REGION Network 2: Block description — Sections 3.2 to 3.4
   // ▂▂▂▂▂▂▂▂▂▂▂▂▂▂▂▂▂▂▂▂▂▂▂▂▂▂▂▂▂▂▂▂▂▂▂▂▂▂▂▂▂▂▂▂
   // 3.2     Warnings and alarms
   // 
   // 
   // By default, the block generates 4 alarms and warnings (2 warnings and 2 alarms, 4 in total) 
   // as follows:
   // 
   // 
   //  ――――――――――――――――――――――――――――――――――――――――――
   //  ALARM / WARNING     FUNCTION
   //  ――――――――――――――――――――――――――――――――――――――――――
   //  Alarm high       Scaled signal is equal to or above a preset alarm high setpoint
   //  Warning high      Scaled signal is equal to or above a preset warning high setpoint
   //  Warning low     Scaled signal is equal to or below a preset warning low setpoint
   //  Alarm low      Scaled signal is equal to or below a preset alarm low setpoint
   //  ――――――――――――――――――――――――――――――――――――――――――
   //  Default alarm and warning signals
   // 
   // 
   // The active state of any alarm or warning is stored in the DYNAMIC_DATA structure in the following 
   // variables:
   // 
   // 
   //  UT22001_Dy_InstAnalogRead
   //  ――――――――――――――――――――――――――――――――――――――――――
   //  SIGNAL NAME          FUNCTION                     TYPE
   //  ――――――――――――――――――――――――――――――――――――――――――
   //  msg_Alm_H         MESSAGE — Alarm - high alarm is active        Bool
   //  msg_Alm_L          MESSAGE — Alarm - low alarm is active          Bool
   //  msg_Wrn_H          MESSAGE — Warning - high warning is active      Bool
   //  msg_Wrn_L          MESSAGE — Warning - low warning is active        Bool
   //  ――――――――――――――――――――――――――――――――――――――――――
   // 
   // 
   // The alarms and warnings that end with _H are activated when the scaled instrument reading is 
   // greater than or equal to a setpoint threshold (i.e. activate when the measured quantity is too 
   // high; generally, if there is both an alarm high and a warning high, the convention within the PAL 
   // is that the warning should activate before the alarm².
   // 
   // 
   // The alarms and warnings that end with _L are activated when the scaled instrument reading is 
   // less than or equal to a setpoint threshold (i.e. activate when the measured quantity is too low; 
   // generally, if there is both an alarm low and a warning low, the convention within the PAL is that 
   // the warning should activate before the alarm².
   // 
   // ――――――――――
   // ²         This is just a convention, there is nothing to stop the warning being set to occur after 
   //      the alarm (i.e. the warning detecting the most extreme condition). All alarms and 
   //      warnings are entirely independent of each other and no error checking is carried 
   //      out to ensure that any particular threshold is above or below another.
   // ――――――――――
   // 
   // All alarms and warnings are individually enabled (a disabled alarm or warning will never be 
   // activated), all alarms and warnings have individual setpoint values (the value at which the 
   // alarm or warning is triggered), all alarms and warnings have individual hysteresis valves 
   // (effectively a tolerance band, the difference between where an alarm activates and where it 
   // deactivates, used to prevent nuisance or “chattering” alarms). Finally, each alarm and warning 
   // has a configurable on and off delay (the alarm or warning will only activate if the reading is 
   // outside the threshold for the on-delay time and similarly will only deactivate when the reading 
   // is inside the threshold and hysteresis for the off-delay time).
   // 
   // The following table summarises all the available signals for each alarm and warning:
   // 
   // 
   //  ――――――――――――――――――――――――――――――――――――――――――
   //  SIGNAL          FUNCTION             TYPE   DETAILS
   //  ――――――――――――――――――――――――――――――――――――――――――
   //  CONFIG_XXX_Y_EN    Alarm/warning enabled      Bool    1 = enabled, 0 = disabled
   //  SP_XXX_Y_VAL      Alarm/warning setpoint value    Real Engineering units
   //  SP_XXX_Y_HYST_VAL    Alarm/warning hysteresis value Real Engineering units
   //  TIME_XXX_Y_ON_DEL   Alarm/warning on delay time   Real In seconds
   //  TIME_XXX_Y_OFF_DEL     Alarm/warning off delay time   Real In seconds
   //  mode_Xxx_Y_MaskOn     Alarm/warning is masked      Bool    1 = masked, 0 = normal
   //  msg_Xxx_Y         Alarm/warning is active      Bool    1 = active, 0 = inactive
   //  ――――――――――――――――――――――――――――――――――――――――――
   //  Default alarm and warning signals — where XXX is either ALM or WRN and Y is either H or L
   // 
   // 
   // 
   // ▁▁▁▁▁▁▁▁▁▁▁▁▁▁▁▁▁▁▁▁▁▁▁▁▁▁▁▁▁▁▁▁▁▁▁▁▁▁▁▁▁▁▁▁
   // 3.2.1     High alarms and warnings (an example)
   // 
   // 
   // This example explains how a high alarm signal is generated, a high warning works in exactly the 
   // same way with WRN being substituted for ALM.
   // 
   // The full set of signals associated with the high alarm are:
   // 
   // 
   //  ――――――――――――――――――――――――――――――――――――――――――
   //  SIGNAL           FUNCTION            TYPE   DETAILS
   //  ――――――――――――――――――――――――――――――――――――――――――
   //  CONFIG_ALM_H_EN    Alarm high enabled      Bool    1 = enabled, 0 = disabled
   //  SP_ALM_H_VAL      Alarm high setpoint value    Real Engineering units
   //  SP_ALM_H_HYST_VAL    Alarm high hysteresis value Real Engineering units
   //  TIME_ALM_H_ON_DEL   Alarm high on delay time   Real In seconds
   //  TIME_ALM_H_OFF_DEL     Alarm high off delay time   Real In seconds
   //  mode_Alm_H_MaskOn    Alarm is masked         Bool    1 = masked, 0 = normal
   //  msg_Alm_H        Alarm high is active      Bool    1 = active, 0 = inactive
   //  ――――――――――――――――――――――――――――――――――――――――――
   // 
   // 
   // The figure below indicates how each of these signal functions (note TIME_ALM_H_ON_DEL and
   // TIME_ALM_H_OFF_DEL have been abbreviated to ON_DEL and OFF_DEL respectively):
   // 
   // 
   //                 │
   //                 │          ╱╲╱╲
   //                 │    ①      ②╱    ╲
   //       SP_ALM_H_VAL↘│____╱╲________╱____________╲③_______④__________ 
   //    SP_ALM_H_HYST_VAL ↕│__╱____╲____╱╎_____╎_______╲____╱╲___________
   //                 │╱    ╲╱ ╎    ╎      ╲╱     ╲
   //                 │        ╎    ╎          ╎╲
   //                 │        ╎    ╎          ╎ ╲___
   //                 │        ╎    ╎          ╎    ╎╲╱
   //                 │    ON_DEL→╎    ╎←    OFF_DEL→╎    ╎←
   //                 ┼─────────────────────────────
   // 
   //                            ╎                        ╎
   // 
   //         msg_Alm_H │             ┏━━━━━━━━━━━━┓
   //                 │             ┃               ┃
   // CONFIG_ALM_H_EN = 1     │             ┃   ALARM IS ACTIVE    ┃
   // & mode_Alm_H_MaskOn = 0 │             ┃               ┃
   //                 │             ┃               ┃
   //                 ┼━━━━━━━━━━━━╶╶╶╶╶╶╶╶╶╶╶╶╶━━━━
   // 
   //                            ╎                        ╎
   // 
   //         msg_Alm_H │          
   // ⑤               │             ╎               ╎             
   // CONFIG_ALM_H_EN = 0     │             
   //     OR          │             ╎               ╎
   // CONFIG_ALM_H_EN = 1     │          
   // & mode_Alm_H_MaskOn = 1 ┼━━━━━━━━━━━━━━━━━━━━━━━━━━━━━
   // 
   // 
   // 
   // ▁▁▁▁▁▁▁▁▁▁▁▁▁▁▁▁▁▁▁▁▁▁▁▁▁▁▁▁▁▁▁▁▁▁▁▁▁▁▁▁▁▁▁▁
   // Scenario ①, alarm setpoint reached, but for less than on-delay duration
   // 
   // 
   // The graph represents the scaled analog instrument reading, actual_Value (in engineering 
   // units). The top horizontal line is the setpoint for the high alarm (SP_ALM_H_VAL).
   // 
   // If the alarm is enabled (CONFIG_ALM_H_EN = 1) then the following actions occur:
   // 
   // At point ① on the graph, the signal actual_Value reaches (and exceeds) the threshold value 
   // SP_ALM_H_VAL; i.e.:
   // 
   //           actual_Value ≥ SP_ALM_H_VAL
   // 
   // At this point, the alarm setpoint is exceeded and the on-delay timer starts; in the case of point ①, 
   // the signal actual_Value falls back below the setpoint value before the on-delay timer reaches 
   // the time set in TIME_ALM_H_ON_DEL, consequently the alarm does not activate.
   // 
   // 
   // 
   // ▁▁▁▁▁▁▁▁▁▁▁▁▁▁▁▁▁▁▁▁▁▁▁▁▁▁▁▁▁▁▁▁▁▁▁▁▁▁▁▁▁▁▁▁
   // Scenario ②, alarm setpoint reached for more than the on-delay duration
   // 
   // 
   // At point ② on the graph, the signal actual_Value again reaches (and exceeds) the setpoint value 
   // SP_ALM_H_VAL.
   // 
   // Again, at this point, the alarm threshold is exceeded and the on-delay timer starts; in the case of 
   // point ②, the signal actual_Value remains at or above the setpoint value for the full duration of 
   // the TIME_ALM_H_ON_DEL and consequently the alarm activates (msg_Alm_H goes to a high 
   // state), this is indicated in the middle msg_Alm_H graph.
   // 
   // 
   // 
   // ▁▁▁▁▁▁▁▁▁▁▁▁▁▁▁▁▁▁▁▁▁▁▁▁▁▁▁▁▁▁▁▁▁▁▁▁▁▁▁▁▁▁▁▁
   // Scenario ③, alarm reset level reached, but for less than the off-delay duration
   // 
   // 
   // At point ③, the signal actual_Value falls to the point at which the alarm is no longer active i.e.:
   // 
   //           actual_Value < (SP_ALM_H_VAL − SP_ALM_H_HYST_VAL)
   // 
   // Note:    in this case the inequality is less than (not less than or equal to), this is to prevent 
   //      conflict detecting the threshold and detecting the reset value if SP_ALM_H_HYST_VAL 
   //      is set to zero.
   // 
   // At this point, the signal is below the alarm reset level:
   // 
   //           SP_ALM_H_VAL − SP_ALM_H_HYST_VAL
   // 
   // and the off-delay timer starts; in the case of point ③, the signal actual_Value returns above the 
   // reset threshold before the off-delay timer reaches the time set in TIME_ALM_H_OFF_DEL, 
   // consequently, the alarm does not deactivate.
   // 
   // 
   // 
   // ▁▁▁▁▁▁▁▁▁▁▁▁▁▁▁▁▁▁▁▁▁▁▁▁▁▁▁▁▁▁▁▁▁▁▁▁▁▁▁▁▁▁▁▁
   // Scenario ④, alarm reset level reached for more than the off-delay duration
   // 
   // 
   // At point ④ on the graph, the signal actual_Value again falls below the alarm reset level 
   // (SP_ALM_H_VAL − SP_ALM_H_HYST_VAL).
   // 
   // Again, at this point, the off-delay timer starts; in the case of point ④, the signal actual_Value 
   // remains below the reset threshold for the full duration of the TIME_ALM_H_OFF_DEL and 
   // consequently, the alarm deactivates (msg_Alm_H goes to a low state), this is indicated in the 
   // middle msg_Alm_H graph.
   // 
   // 
   // 
   // ▁▁▁▁▁▁▁▁▁▁▁▁▁▁▁▁▁▁▁▁▁▁▁▁▁▁▁▁▁▁▁▁▁▁▁▁▁▁▁▁▁▁▁▁
   // Scenario ⑤, alarm is disabled
   // 
   // 
   // If the alarm is disabled (CONFIG_ALM_H_EN = 0) then the alarm will never activate 
   // (msg_Alm_H is always in a low state), this is indicated in the lower msg_Alm_H graph.
   // 
   // Note:    The timer for disabled alarms and warnings is permanently set to zero.
   // 
   // 
   // ▁▁▁▁▁▁▁▁▁▁▁▁▁▁▁▁▁▁▁▁▁▁▁▁▁▁▁▁▁▁▁▁▁▁▁▁▁▁▁▁▁▁▁▁
   // 3.2.2     Low alarms and warnings
   // 
   // 
   // Low alarms and warnings are very similar to the high alarms of § 3.2.1, they do however work
   // in the opposite sense (the inequalities are reversed), low alarms and warnings are activated
   // when the actual_Value falls below, or is equal to, the SP_ALM_L_VAL, and deactivates when it
   // rises above SP_ALM_L_VAL + SP_ALM_L_HYST_VAL.
   // 
   // On and off delays work in exactly the same way as those for the high alarm.
   // 
   // A worked example of the low alarm is given in the online documentation for this block:
   // 
   // select this block in the project tree and press:
   //      SHIFT + F1 or follow the link: https://psop.uk/pal-smds-fc02001-p
   // 
   // 
   // 
   // 
   // ▁▁▁▁▁▁▁▁▁▁▁▁▁▁▁▁▁▁▁▁▁▁▁▁▁▁▁▁▁▁▁▁▁▁▁▁▁▁▁▁▁▁▁▁
   // 3.2.3     Masking alarms and warnings
   // 
   // 
   // There are conditions where it can become necessary to mask (supress) alarms and warnings, a 
   // typical example could be a flow meter that monitors the flow into a filter; under normal 
   // conditions the flow meter would generate a low alarm if the flow into the filter were below a 
   // certain setpoint (indicating that the filter is becoming blocked).
   // 
   // It would be normal practice to supress this alarm when the filter was being cleaned, under 
   // these circumstances there would be no flow into the filter, but this would be a normal operating 
   // condition for the filter; the flow meter should only be monitoring for a low alarm during normal 
   // operation, not when the filter is being cleaned.
   // 
   // This suppression of an alarm or warning is referred to as “masking”, and there is a mask bit for 
   // each alarm and warning:
   // 
   // 
   //  ――――――――――――――――――――――――――――――――――――――――――
   //  SIGNAL           FUNCTION           TYPE   DETAILS
   //  ――――――――――――――――――――――――――――――――――――――――――
   //  mode_Alm_H_MaskOn    Masks the high alarm     Bool    1 = alarm masked, 0 = normal
   //  mode_Alm_L_MaskOn    Masks the low alarm    Bool    1 = alarm masked, 0 = normal
   //  mode_Wrn_H_MaskOn    Masks the high warning    Bool    1 = warning masked, 0 = normal
   //  mode_Wrn_L_MaskOn     Masks the low warning      Bool    1 = warning masked, 0 = normal
   //  ――――――――――――――――――――――――――――――――――――――――――
   //  Alarm and warning mask signals
   // 
   //  
   // Any alarm or warning that is masked (mode_Xxx_Y_MaskOn = 1), will deactivate instantly 
   // (there is no off-delay) and will not reactivate activate (the msg_Xxx_Y will be set to zero), the 
   // effect is the same as if the CONFIG_XXX_Y_EN bit were turned off.
   // 
   // The difference between the mask and the ENABLE signals is that the enable signal is a 
   // configuration of the instrument (it determines which alarms and warnings are configured for the 
   // particular instrument) and does not change at run-time (it is stored in static data block).
   // 
   // The mask signal on the other hand can be changed at run-time (either by some aspect of the 
   // Controller program or by the operator). The mask signal is stored in a dynamic data block and 
   // can be freely modified.
   // 
   // Note:    If an alarm or warning is not enabled (CONFIG_XXX_Y_EN = 0), then the mask bit 
   //      (mode_Xxx_Y_MaskOn) will not do anything (setting it will not enable the alarm), in 
   //      fact if the alarm or warning is not enabled, the mask bit will be permanently set to 
   //      zero.
   // 
   // Masking alarms and warnings is the correct way to disable an alarm as part of the process 
   // operation of the plant.
   // 
   // When an alarm or warning goes from a masked condition to an unmasked condition (returns to 
   // normal operation), the on-delay timer will be reset and any alarm or warning condition will 
   // have to go back through the on-delay process before the alarm or warning can reactivate, this is 
   // true even if the alarm were active before being masked.
   // 
   // 
   // 
   // 
   // ▁▁▁▁▁▁▁▁▁▁▁▁▁▁▁▁▁▁▁▁▁▁▁▁▁▁▁▁▁▁▁▁▁▁▁▁▁▁▁▁▁▁▁▁
   // 3.2.4     A note on dynamically enabling alarms
   // 
   // 
   // In normal operations, alarms are either enabled or disabled as part of the instrument 
   // configuration and this configuration will not change during run-time; the enable signal 
   // (CONFIG_XXX_Y_EN) is after all in a static data block. 
   // 
   // However, it is possible that the static data block is being used as a recipe block and as such it 
   // could be overloaded at some point during run-time.
   // 
   // Should the block detect a change in any of the CONFIG_XXX_Y_EN; specifically, a rising 
   // edge, the block provides error checking to ensure that the associated alarm/warning timer 
   // (actual_Xxx_Y_Timer) is preset to correct TIME_XXX_Y_ON_DEL, this prevents the alarm/warning 
   // from activating instantly, if the actual_Value is outside the alarm/warning setpoint. A condition 
   // that could arise because the timer is set to zero while ever the alarm/warning is disabled.
   // 
   // Note:    This is a minor technical point, but it is a necessary error trapping mechanism — the 
   //      situation could arise even if it is unlikely.
   // 
   // 
   // 
   // ▂▂▂▂▂▂▂▂▂▂▂▂▂▂▂▂▂▂▂▂▂▂▂▂▂▂▂▂▂▂▂▂▂▂▂▂▂▂▂▂▂▂▂▂
   // 3.3     Fault signals
   // 
   // 
   // There are four fault signals that can be produced by the block:
   // 
   // 
   //  ――――――――――――――――――――――――――――――――――――――――――
   //  SIGNAL           FUNCTION            TYPE   DETAILS
   //  ――――――――――――――――――――――――――――――――――――――――――
   //  msg_Flt_UnderRange   The instrument is more than   Bool    1 = under-range, 0 = healthy
   //                 a percentage below the its 
   //                 minimum value
   // 
   //  msg_Flt_OverRange     The instrument is more than   Bool    1 = over-range, 0 = healthy
   //                 a percentage above its 
   //                 maximum value
   // 
   //  msg_Flt_OutOfRange   Common fault, either       Bool    1 = out-of-range, 0 = healthy
   //                 under or over range
   // 
   //  msg_Flt_External     The instrument itself is    Bool    1 = fault, 0 = healthy
   //                 indicating a fault 
   //                 (hardwired signal)
   //  ――――――――――――――――――――――――――――――――――――――――――
   //  Block fault signals 
   // 
   // 
   // 
   // ▁▁▁▁▁▁▁▁▁▁▁▁▁▁▁▁▁▁▁▁▁▁▁▁▁▁▁▁▁▁▁▁▁▁▁▁▁▁▁▁▁▁▁▁
   // 3.3.1     Over, under and out of range fault signals
   // 
   // If the scaled signal actual_Value , is outside the RANGE_SCALE_MIN to RANGE_SCALE_MAX range 
   // (dotted area of the graph, § 3.1), the scaled instrument reading (actual_Value) will still be 
   // calculated correctly; however, an appropriate, over-range or under-range (msg_Flt_OverRange or 
   // msg_Flt_UnderRange) signal will be generated to indicate that the instrument signal is outside 
   // of its calibrated range and is potentially no longer accurate.
   // 
   // Some tolerance is permitted before either the msg_Flt_OverRange or msg_Flt_UnderRange 
   // signals is activated (this is to prevent nuisance alarms — most instruments are tolerant of slight 
   // over and under shoot readings). 
   // 
   // The tolerance applied to the out-of-range signals is a percentage of the scaled range of the 
   // instrument (the scaled range being RANGE_SCALE_MAX − RANGE_SCALE_MIN). 
   // 
   // The tolerance to be applied is given in the parameter RANGE_OOR_PERCENT, this is a real 
   // (floating point) number in the range 0.0-10.0%.
   // 
   // If the tolerance for the instrument is not known, a generic value of 2.5% should be used.
   // 
   // The out-of-range tolerance absolute value (in terms of the actual_Value rather than as a 
   // percentage) is calculated as:
   // 
   // 
   // ┌───────────────────────────────────────┐
   // │                            (RANGE_SCALE_MAX ─ RANGE_SCALE_MIN) ╳ RANGE_OOR_PERCENT  │
   // │ calAbsOOR =  ――――――――――――――――――――――――――――――    │
   // │                        100                 │
   // └───────────────────────────────────────┘
   // 
   // 
   // Thus, if RANGE_SCALE_MIN is −100 l/s, RANGE_SCALE_MAX is +100 l/s (giving a span of 200 l/s) and 
   // a RANGE_OOR_PERCENT of 2.5% is selected, the absolute out of range value (calAbsOOR in the 
   // above equation) has a calculated value of 5.00 l/s (2.5% of 200).
   // 
   // In this example, the msg_Flt_OverRange signal would activate when actual_Value exceeded a 
   // value of RANGE_SCALE_MAX + 5.00 (or 105.00  l/s). This value (the absolute over range limit 
   // value) is stored in a calculated variable cal_OR_Abs. 
   // 
   // Similarly, the msg_Flt_UnderRange signal would activate when actual_Value fell below a value 
   // of RANGE_SCALE_MIN – 5.00 (or −105.00  l/s). This value (the absolute under range limit value) 
   // is stored in a calculated variable cal_UR_Abs.
   // 
   // Both the cal_OR_Abs and cal_UR_Abs values are stored in  the dynamic data area and can be 
   // accessed by SCADA and HMI systems, or other aspects of the Con-troller software.
   // 
   // 
   // 
   // ▁▁▁▁▁▁▁▁▁▁▁▁▁▁▁▁▁▁▁▁▁▁▁▁▁▁▁▁▁▁▁▁▁▁▁▁▁▁▁▁▁▁▁▁
   // Common out of range signal
   // 
   // 
   // There is a third out of range signal: msg_Flt_OutOfRange, this signal is a common signal that 
   // just indicates the instrument is out of its calibrated range (it does not specify whether it is over 
   // or under range). It is activated if either the msg_Flt_OverRange or msg_Flt_UnderRange signal is 
   // active.
   // 
   // 
   // 
   // ▁▁▁▁▁▁▁▁▁▁▁▁▁▁▁▁▁▁▁▁▁▁▁▁▁▁▁▁▁▁▁▁▁▁▁▁▁▁▁▁▁▁▁▁
   // Configuration error
   // 
   // If a range configuration error is present (see § 3.1.2), all three out of range signals will activate 
   // msg_Flt_OverRange, msg_Flt_UnderRange and msg_Flt_OutOfRange.
   // 
   // 
   // 
   // ▁▁▁▁▁▁▁▁▁▁▁▁▁▁▁▁▁▁▁▁▁▁▁▁▁▁▁▁▁▁▁▁▁▁▁▁▁▁▁▁▁▁▁▁
   // 3.3.2     External fault signal
   // 
   // 
   // The external fault is an optional hardwired signal from the instrument, it indicates that the 
   // instrument itself is registering that there is some problem. Such external fault signals are more 
   // commonly associated with complex instruments (mass flow metres, ultrasonic level 
   // transducers, analytical instruments &c.) rather than the more simplistic instruments (pressure 
   // sensors, temperature transmitters &c.).
   // 
   // Typical examples of external faults would be:
   // 
   //    •   No medium present in a mass flow meter (if the instrument were measuring liquid 
   //      flow and the pipe had become empty)
   // 
   //    •   Foam indication from an ultrasonic level transducer (preventing an accurate level 
   //      reading)
   // 
   // Such fault signals are generally indicated via a hardwired digital input to the Controller.
   // 
   // The external fault signal (if used) is passed to the block as the parameter: EXT_FAULT
   // 
   // 
   //  ――――――――――――――――――――――――――――――――――――――――――
   //  PARAMETER          FUNCTION            TYPE   DETAILS
   //  ――――――――――――――――――――――――――――――――――――――――――
   //  EXT_FAULT        Hardwired signal indicating    Bool    1 = fault, 0 = healthy
   //                 the instrument is in a fault 
   //                 condition
   //  ――――――――――――――――――――――――――――――――――――――――――
   //  Block external fault parameter 
   // 
   // 
   // If the EXT_FAULT signal is not required, the input should be set to _false.
   // 
   // If the instrument generates a fault signal in the opposite sense, i.e. 0 = fault and 1 = healthy (this 
   // is a common fail-safe condition, that generates a fault signal if the instrument is disconnected 
   // or a wire break occurs), then a normally closed contact should be applied to the EXT_FAULT 
   // parameter to invert the signal into the block (see below):
   // 
   // 
   //                            ┌─────────────
   //         ───────────────────┤ FC02001 
   //                            │               │                       
   //                                "FC001" ─┤ AI_RAW_SIGNAL          │
   //                            │               │
   //       "DB00801_St_ConstAiRawData".AI_RAW_2003 ─┤ AI_RAW_DATA           │
   //                            │               │
   //    "DB00851_St_ConstAiScaleData".AI_SCALE_FC001    ─┤ AI_SCALE_DATA          │
   //                            │               │
   //              "FC001_FAULT"           │               │
   //           ────┤╱├──────────┤ EXT_FAULT                │
   //                            │               │
   //                            │               │
   //         "DB02001_St_StdInstAnalogRead".FC001 ─┤ STATIC_DATA             │
   //                            │
   //        "DB22001_Dy_StdInstAnalogRead".FC001 ─┤ DYNAMIC_DATA
   //                            │
   //                            │
   // 
   // 
   // If the EXT_FAULT parameter is activated (set to 1), the corresponding fault signal within the 
   // dynamic data (msg_Flt_External) will be activated, there are no delays or other filtering 
   // associated with this signal.
   // 
   // Note:    The external fault does not in any way impact the reading and scaling of the 
   //      instrument or the production of any alarms or warnings.
   // 
   // 
   // 
   // ▂▂▂▂▂▂▂▂▂▂▂▂▂▂▂▂▂▂▂▂▂▂▂▂▂▂▂▂▂▂▂▂▂▂▂▂▂▂▂▂▂▂▂▂
   // 3.4     Operating mode
   // 
   // 
   // This block  supports various operating modes:
   // 
   //    •   Simulation mode
   //    •   Remote/local mode
   //    •   Faceplate disabled mode
   // 
   // Examining these in turn:
   // 
   // 
   // ▁▁▁▁▁▁▁▁▁▁▁▁▁▁▁▁▁▁▁▁▁▁▁▁▁▁▁▁▁▁▁▁▁▁▁▁▁▁▁▁▁▁▁▁
   // 3.4.1     Simulation mode
   // 
   // 
   // The instrument can be switched to a simulation mode, in which the actual reading from the 
   // instrument is replaced by a simulated value provided by the operator. 
   // 
   // Simulation mode is generally used during testing, but can also be applied in a process 
   // environment if a fault condition is detected within the instrument; this scenario allows the plant 
   // to continue operating (albeit under some degree of manual control) until the instrument is 
   // repaired or replaced.
   // 
   // The following data points are associated with the simulation mode:
   // 
   // 
   //  ――――――――――――――――――――――――――――――――――――――――――
   //  SIGNAL           FUNCTION            TYPE   DETAILS
   //  ――――――――――――――――――――――――――――――――――――――――――
   //  CONFIG_SIM_DIS         Prevents simulation mode   Bool    1 = no sim, 0 = sim permitted
   //                 being activated under all 
   //                 circumstances
   // 
   //  mode_SimOn        Activates simulation mode,    Bool    1 = sim on, 0 = sim off
   //                 if active, the scaled reading 
   //                 of the instrument:
   //                 actual_Value will be set 
   //                 to mode_SimValue
   // 
   //  mode_SimValue      Scaled instrument reading   Real    Simulated instrument value
   //                 actual_Value will be set to  
   //                 this if simulation mode is 
   //                 on (CONFIG_SIM_DIS = 0 
   //                 and mode_SimOn = 1)
   // 
   //  status_SimOn       Status indication, shows if    Bool    1 = sim active, 0 = Sim off
   //                 simulation mode is active
   //  ――――――――――――――――――――――――――――――――――――――――――
   // 
   // 
   // Simulation mode can only be activated by the operator via a faceplate available at the 
   // supervisory system (SCADA/HMI).
   // 
   // If simulation mode is disabled (configuration signal CONFIG_SIM_DIS is set to 1), then the 
   // simulation mode cannot be turned on under any circumstances, the option is greyed out on the 
   // supervisory system faceplate and the block will constantly reset the mode_SimOn signal.
   // 
   // If simulation mode is permitted (CONFIG_SIM_DIS = 0), then setting mode_SimOn to 1 will 
   // activate simulation mode and the scaled instrument value (actual_Value) will be set to the 
   // value stored in mode_SimValue:
   // 
   //           i.e. actual_Value = mode_SimValue
   // 
   // and all fault messages will be reset.
   // 
   // The operator can set and adjust the simulation value (mode_SimValue) from the instrument
   // faceplate on the supervisory system. The simulation value can be adjusted at any time by the 
   // operator (even if simulation mode has not been activated), but will not be applied until 
   // simulation mode is turned on (mode_SimOn = 1). 
   // 
   // If simulation mode is completely disabled (CONFIG_SIM_DIS is set to 1) then the operator will
   // not be able to adjust the simulated value (mode_SimValue will be greyed out on the faceplate).
   // 
   // 
   // 
   // ▁▁▁▁▁▁▁▁▁▁▁▁▁▁▁▁▁▁▁▁▁▁▁▁▁▁▁▁▁▁▁▁▁▁▁▁▁▁▁▁▁▁▁▁
   // 3.4.2     Remote/local mode
   // 
   // 
   // Remote and local operating modes refer to the supervisory system that has control of the 
   // instrument (i.e. which system can write to the device and change the operating mode of the 
   // device). 
   // 
   // This type of mode is usual present where a plant has a remote central control location (a control 
   // room) that normally controls the device (remote control), but also has a field panel with a local 
   // HMI that an operator in the field can select to take over control of the device (local control) for 
   // maintenance purposes.
   // 
   // The modes are as follows (and are mutually exclusive, only one will be active):
   // 
   //    Remote        Only the remote system in the control room can 
   //                 control the device
   // 
   //    Local            A local system has taken control of the device and the remote 
   //                 system can no longer issue commands to it
   // 
   //    Remote/local disabled   The system does not use remote/local modes and any 
   //    (ALL mode)       supervisory system can issue commands to the device 
   //  
   // Remote/local control is generally handled by the supervisory systems themselves; however, the 
   // supervisory systems need a storage area per device to record which mode that device is in, local 
   // control is often activated by a panel key-switch, that changes the state of several devices from 
   // remote to local (usually all the devices controlled by the local panel).
   // 
   // The block simply identifies the remote/local mode from the mode signals and configuration 
   // signals provided to the block.
   // 
   // For systems that do not use remote/local modes (any supervisory system can control the device, 
   // or control is determined by operator privileges), the remote/local modes can be disabled 
   // (CONFIG_RL_EN is set to zero) and the device is effectively in ALL mode (any system can 
   // control the device).
   // 
   // If remote/local operation is in use, the supervisory system that does not have control will still 
   // display all the information from the device, but will not be able to control the device (it could not 
   // for example, activate simulation mode) and all control function (faceplate functions) will be 
   // greyed out.
   // 
   // The following signals are associated with remote/local/all modes:
   // 
   // 
   //  ――――――――――――――――――――――――――――――――――――――――――
   //  SIGNAL           FUNCTION            TYPE   DETAILS
   //  ――――――――――――――――――――――――――――――――――――――――――
   //  CONFIG_RL_EN      Allows Remote and Local      Bool    1 = Remote/local selected
   //                 modes to be selected        0 = All mode is active
   // 
   //  mode_RemoteOn       Activates remote mode     Bool    1 = remote mode on, 
   //                 CONFIG_RL_EN must = 1       0 = remote mode off
   // 
   //  mode_LocalOn     Activates local mode          Bool    1 = local mode on, 
   //                 CONFIG_RL_EN must = 1       0 = remote mode off
   // 
   //  status_RemoteOn      Status remote mode on     Bool    1 = remote mode on, 
   //                               0 = remote mode off
   // 
   //  status_LocalOn       Status local mode on      Bool    1 = local mode on, 
   //                               0 = local mode off
   // 
   //  status_RLOff       Status Remote/local is off     Bool    1 = ALL mode on, 
   //              (ALL mode active)         0 = ALL mode off
   //  ――――――――――――――――――――――――――――――――――――――――――
   //  Block remote/local signals 
   // 
   // 
   // By default, remote/local is disabled — ALL mode is selected (CONFIG_RL_EN = 0).
   // 
   // 
   // 
   // 
   // ▁▁▁▁▁▁▁▁▁▁▁▁▁▁▁▁▁▁▁▁▁▁▁▁▁▁▁▁▁▁▁▁▁▁▁▁▁▁▁▁▁▁▁▁
   // 3.4.3     Faceplate disable mode
   // 
   // 
   // It is possible to disable the supervisory system faceplate from within the block, the configuration 
   // signal:
   // 
   // 
   //  ――――――――――――――――――――――――――――――――――――――――――
   //  SIGNAL           FUNCTION            TYPE   DETAILS
   //  ――――――――――――――――――――――――――――――――――――――――――
   //  CONFIG_FP_DIS        Disable the supervisory      Bool    1 = Faceplate disabled
   //                 system faceplate           0 = normal
   //  ――――――――――――――――――――――――――――――――――――――――――
   //  Block faceplate disable signal 
   // 
   // 
   // If the faceplate is disabled (CONFIG_FP_DIS = 1), the supervisory system will not allow the 
   // device faceplate to be opened (normally achieved by clicking the block icon or device symbol), 
   // this in turn prevents the operator from affecting the device in anyway, it would not, for example, 
   // be possible to put the device into simulation mode.
END_REGION

REGION Network 3: Block description — Sections 3.5 to 11
   // ▂▂▂▂▂▂▂▂▂▂▂▂▂▂▂▂▂▂▂▂▂▂▂▂▂▂▂▂▂▂▂▂▂▂▂▂▂▂▂▂▂▂▂▂
   // 3.5     Status reporting
   // 
   // The module constantly reports the status of the instrument (i.e. alarm/warning states, faults &c.) 
   // via various status signals. These signals can be used within the Controller software to determine 
   // specific device conditions (e.g. a high alarm is active), the signals may also be used by 
   // supervisory systems to display (in an ani-mated fashion) the state of the instrument.
   // 
   // The status signals for faults, alarms and warnings are either duplicates of the message signals 
   // (signals beginning with msg_) or logical combinations of them.
   // 
   // The following is a full list of the status signals:
   // 
   // 
   //  UT22001_Dy_InstAnalogRead
   //  ――――――――――――――――――――――――――――――――――――――――――
   //  SIGNAL           FUNCTION            TYPE   DETAILS
   //  ――――――――――――――――――――――――――――――――――――――――――
   //  status_Alm_H        Identical to: msg_Alm_H    Bool    1 = high alm active, 0 = no alm
   // 
   //  status_Alm_L         Identical to: msg_Alm_L       Bool    1 = low alm active, 0 = no alm
   // 
   //  status_Wrn_H        Identical to: msg_Wrn_H    Bool    1 = high wrn active, 0 = no wrn
   // 
   //  status_Wrn_L         Identical to: msg_Wrn_L     Bool    1 = low wrn active, 0 = no wrn
   // 
   //  status_Alm_H_Mask     High alarm is masked     Bool    1 = masked, 0 = normal
   // 
   //  status_Alm_L_Mask   Low alarm is masked      Bool    1 = masked, 0 = normal
   // 
   //  status_Wrn_H_Mask      High warning is masked    Bool    1 = masked, 0 = normal
   // 
   //  status_Wrn_L_Mask       Low warning is masked     Bool    1 = masked, 0 = normal
   // 
   //  status_Alm_H_Dis         High alarm is disabled       Bool    1 = disabled, 0 = normal
   // 
   //  status_Alm_L_Dis       Low alarm is disabled        Bool    1 = disabled, 0 = normal
   // 
   //  status_Wrn_H_Dis          High warning is disabled      Bool    1 = disabled, 0 = normal
   // 
   //  status_Wrn_L_Dis           Low warning is disabled       Bool    1 = disabled, 0 = normal
   // 
   //  status_Fault       Indicates any of the msg_Flt    Bool    1 = fault active, 0 = healthy
   //                 signals are active:
   //                  msg_Flt_UnderRange
   //                  msg_Flt_OverRange
   //                  msg_Flt_OutOfRange
   //                  msg_Flt_External 
   // 
   //  status_SimOn       Status simulation mode on     Bool    1 = sim on, 0 = sim off
   // 
   //  status_RemoteOn      Status remote mode on     Bool    1 = rem on, 0 = rem off
   // 
   //  status_LocalOn       Status local mode on      Bool    1 = loc on, 0 = loc off 
   // 
   //  status_RLOff       Status ALL mode is on           Bool    1 = ALL mode on, 
   //                               0 = ALL mode off
   //  ――――――――――――――――――――――――――――――――――――――――――
   //  Block status signals 
   // 
   // 
   // 
   // ▁▁▁▁▁▁▁▁▁▁▁▁▁▁▁▁▁▁▁▁▁▁▁▁▁▁▁▁▁▁▁▁▁▁▁▁▁▁▁▁▁▁▁▁
   // 3.5.1     String constants for tag name and units
   // 
   // 
   // The STATIC_DATA structure holds two string values:
   // 
   // 
   //  UT02001_St_InstAnalogRead
   //  ――――――――――――――――――――――――――――――――――――――――――
   //  SIGNAL NAME          FUNCTION                     TYPE
   //  ――――――――――――――――――――――――――――――――――――――――――
   //  INFO_TAG          INFORMATION — Instrument ID tag          String[20]
   // 
   //  INFO_UNITS          INFORMATION — Instrument engineering units       String[10]
   //                        (unit of measure)
   //  ――――――――――――――――――――――――――――――――――――――――――
   //  String constants for the instrument
   // 
   // 
   // These two strings allow the supervisory system to populate the instrument tag (e.g. FIC001) and 
   // the engineering units applicable to the instrument (L/s for example) directly from the data 
   // stored in the PLC; it means the block icon can be used directly within the supervisory system 
   // graphic without customisation; all the data will be populated directly at runtime.
   // 
   //                ━━━   ⬙⬙⬙⬙⬙⬙   ━━━
   // 
   // 
   // 
   // ▄▄▄▄▄▄▄▄▄▄▄▄▄▄▄▄▄▄▄▄▄▄▄▄▄▄▄▄▄▄▄▄▄▄▄▄▄▄▄▄▄▄▄▄
   // 4.     Supervisory system interface
   // 
   // 
   // See the online documentation for this block — select the block in the project tree and press:
   //      SHIFT + F1 or follow the link: https://psop.uk/pal-smds-fc02001-p 
   // 
   // An explanation of the block icons and faceplates available to the supervisory system for this 
   // module is given in section 4 of the SMDS document [Ref. 011].
   // 
   // A downloadable copy of the SMDS (and all other project documentation) is available here:
   // 
   //      https://practicalseries.com/2001-pal/21-project/01-00-docs.html
   // 
   // For this module, the document number is: PS2001-5-2312-fc02001
   // 
   //                ━━━   ⬙⬙⬙⬙⬙⬙   ━━━
   // 
   // 
   // 
   // ▄▄▄▄▄▄▄▄▄▄▄▄▄▄▄▄▄▄▄▄▄▄▄▄▄▄▄▄▄▄▄▄▄▄▄▄▄▄▄▄▄▄▄▄
   // 5.     PARAMETERS
   // 
   // 
   // The following parameters are associated with the block:
   // 
   //  
   //  ――――――――――――――――――――――――――――――――――――――――――
   //  PARAM         FUNCTION                      TYPE      IN-OUT 
   //  ――――――――――――――――――――――――――――――――――――――――――
   //  SYS_SIGNALS      Common system signals                UT21000    In
   //           logic and timing signals for parametric access
   // 
   //  AI_RAW_SIGNAL      The unscaled analog input (input word          Word     In
   //           address for the IO card to which the instrument 
   //           is connected)
   //  AI_RAW_DATA      Analog input signal configuration data (type,     UT00801    In
   //           range, descriptions card parameters and 
   //           coefficients)
   // 
   //  AI_SCALE_DATA     Analog input signal scaled value data (instrument   UT00851   In
   //           tag, range, descriptions and engineering units)
   // 
   // 
   //  EXT_FAULT     Optional external fault signal for the instrument     Bool      In
   //           (1 = fault, 0 = healthy). If not required, set 
   //           permanently to _False
   // 
   //  STATIC_DATA     Data structure that holds the configuration data    UT02001    In
   //           for the instrument (raw range, scaled range 
   //           alarm and warning values, filtering times, 
   //           hysteresis values &c.)
   // 
   //  DYNAMIC_DATA      Data structure that holds the live data for the      UT22001    InOut
   //           instrument (its reading in engineering units, 
   //           any alarms or warnings that may be active, 
   //           current timer values, selected operating 
   //           mode &c.)
   //  ――――――――――――――――――――――――――――――――――――――――――
   // 
   // 
   //                ━━━   ⬙⬙⬙⬙⬙⬙   ━━━
   // 
   // 
   // 
   // ▄▄▄▄▄▄▄▄▄▄▄▄▄▄▄▄▄▄▄▄▄▄▄▄▄▄▄▄▄▄▄▄▄▄▄▄▄▄▄▄▄▄▄▄
   // 6.     DATA STRUCTURES AND USAGE
   // 
   // 
   // The block has the following associated data structure:
   // 
   // 
   //  ――――――――――――――――――――――――――――――――――――――――――
   //  DATA STRUCTURE             DESCRIPTION
   //  ――――――――――――――――――――――――――――――――――――――――――
   //  UT01000_St_SysRevision          Revision information for this block    See FC01001
   //  UT01001_St_SysLicence           Licence information for this block  See FC01001
   //  UT21000_Dy_SysSignals           System signals for logic and timing  See FC01001
   // 
   //  UT00801_St_ConstAiRawData        Analog input signal configuration data 
   //                     (type, range, descriptions card parameters and 
   //                     coefficients)
   // 
   //  UT00851_St_ConstAiScaleData     Analog input signal scaled value data 
   //                     (instrument tag, range, descriptions and 
   //                     engineering units)
   // 
   //  UT02001_St_InstAnalogRead      Static data structure for an analog instrument.
   //                     Holds configuration information, instrument ranges 
   //                     and scaling, alarm/warning thresholds &c.
   // 
   //  UT22001_Dy_InstAnalogRead        Dynamic data structure for an analog instrument.
   //                     Current scaled instrument reading, alarm status, 
   //                     operating modes, timer values &c.
   //  ――――――――――――――――――――――――――――――――――――――――――
   // 
   // 
   // 
   // ▂▂▂▂▂▂▂▂▂▂▂▂▂▂▂▂▂▂▂▂▂▂▂▂▂▂▂▂▂▂▂▂▂▂▂▂▂▂▂▂▂▂▂▂
   // 6.1     UT00801_St_ConstAiRawData
   // 
   // 
   // The static data structure for an analog instrument.
   // 
   // 
   //  UT00801_St_ConstAiRawData (full contents)
   //  ―――――――――――――――――――――――――――――――――――――――――― 
   //  SIGNAL NAME          FUNCTION                     TYPE
   //  ――――――――――――――――――――――――――――――――――――――――――
   //  AI_CODE            A 16-bit hex value that uniquely identifies dataset   UInt
   //               (it is the variable name of the dataset in DB00801)
   //  RAW_MIN         Minimum value of the raw analog signal        Int
   //               (at the card)
   // 
   //  RAW_MAX           Maximum value of the raw analog signal        Int
   //  RAW_DESC         Textual plain English description of the channel     String[60]
   //               type and range
   //  PARAM_TYPE         An 8-bit hex code that represents the input type    Byte
   //               See [Ref. 101]
   // 
   //  PARAM_RANGE        An 8-bit hex code that represents the input range    Byte
   //               See [Ref. 101]
   // 
   //  PARAM_COEF        An 8-bit hex code that represents a thermal        Byte
   //               coefficient (thermal resistance channels only, 
   //               otherwise set to 0). See [Ref. 101]
   // 
   //  VALUE_COEF        The actual value of the temperature coefficient in    Real
   //               use (thermal resistance channels only)
   //  ―――――――――――――――――――――――――――――――――――――――――― 
   // 
   // 
   // 
   // ▂▂▂▂▂▂▂▂▂▂▂▂▂▂▂▂▂▂▂▂▂▂▂▂▂▂▂▂▂▂▂▂▂▂▂▂▂▂▂▂▂▂▂▂
   // 6.2     UT00851_St_ConstAiScaleData
   // 
   // 
   // The static data structure for an analog instrument.
   // 
   // 
   //  UT00801_St_ConstAiRawData (full contents)
   //  ―――――――――――――――――――――――――――――――――――――――――― 
   //  SIGNAL NAME          FUNCTION                     TYPE
   //  ――――――――――――――――――――――――――――――――――――――――――
   //  AI_TAG          Tag name of the instrument             UInt
   //  SCALE_MIN        Minimum value of the scaled input signal range    Real
   //               being used by the module
   //  SCALE_MAX          Maximum value of the scaled input signal range      Real
   //               being used by the module
   //  SCALE_UNITS          Engineering units for the instrument         String[20]
   //  SCALE_DESC           Textual plain English description of the instrument  String[60]
   // 
   //  ―――――――――――――――――――――――――――――――――――――――――― 
   // 
   // 
   // 
   // ▂▂▂▂▂▂▂▂▂▂▂▂▂▂▂▂▂▂▂▂▂▂▂▂▂▂▂▂▂▂▂▂▂▂▂▂▂▂▂▂▂▂▂▂
   // 6.3     UT02001_St_InstAnalogRead
   // 
   // 
   // The static data structure for an analog instrument.
   // 
   // 
   //  UT02001_St_InstAnalogRead (full contents)
   //  ―――――――――――――――――――――――――――――――――――――――――― 
   //  SIGNAL NAME          FUNCTION                     TYPE
   //  ―――――――――――――――――――――――――――――――――――――――――― 
   //  CONFIG_ALM_H_EN     CONFIG — High alarm is enabled          Bool
   //                      (1 = enabled, 0 = no alarm) 
   //  CONFIG_ALM_L_EN      CONFIG — Low alarm is enabled           Bool
   //                      (1 = enabled, 0 = no alarm)
   //  CONFIG_WRN_H_EN        CONFIG — High warning is enabled         Bool
   //                      (1 = enabled, 0 = no warning)
   //  CONFIG_WRN_L_EN        CONFIG — Low warning is enabled          Bool
   //                      (1 = enabled, 0 = no warning)
   //  CONFIG_FP_DIS         CONFIG — Faceplate is disabled           Bool
   //                      (1 = no Faceplate, 0 = normal)
   //  CONFIG_SIM_DIS       CONFIG — Simulation is disabled            Bool
   //                      (1 = no Simulation, 0 = normal)
   //  CONFIG_RL_EN       CONFIG — Remote/local mode enabled       Bool
   //                      (1 = enabled, 0 = all mode)
   // 
   //  RANGE_RAW_MIN       RANGE — Minimum value of the raw analog      Int
   //                     signal (at the card). Only used if 
   //                     AI_RAW_DATA is set to User Defined input 
   //                     (AI_CODE = 0000)
   //  RANGE_RAW_MAX      RANGE — Maximum value of the raw analog        Int
   //                     signal (at the card). Only used if 
   //                     AI_RAW_DATA is set to User Defined input 
   //                     (AI_CODE = 0000)
   //  RANGE_OOR_PERCENT      RANGE — Out of range percentage, beyond which    Real
   //                     the instrument is out of range
   // 
   //  SP_ALM_H_VAL       SETPOINT — High alarm threshold value         Real
   //                      [engineering units]
   //  SP_ALM_L_VAL       SETPOINT — Low alarm threshold value       Real
   //                      [engineering units]
   //  SP_WRN_H_VAL         SETPOINT — High warning threshold value        Real
   //                      [engineering units]
   //  SP_WRN_L_VAL       SETPOINT — Low warning threshold value      Real
   //                      [engineering units]
   //  SP_ALM_H_HYST_VAL     SETPOINT — High alarm hysteresis value        Real
   //                      [engineering units]
   //  SP_ALM_L_HYST_VAL     SETPOINT — Low alarm hysteresis value         Real
   //                      [engineering units]
   //  SP_WRN_H_HYST_VAL    SETPOINT — High warning hysteresis value       Real
   //                      [engineering units]
   //  SP_WRN_L_HYST_VAL     SETPOINT — Low warning hysteresis value        Real
   //                      [engineering units]
   // 
   //  TIME_ALM_H_ON_DEL    TIMER — High alarm on delay time          Real
   //                      (activation delay), [seconds]
   //  TIME_ALM_L_ON_DEL     TIMER — Low alarm on delay time           Real
   //                      (activation delay), [seconds]
   //  TIME_WRN_H_ON_DEL       TIMER — High warning on delay time         Real
   //                      (activation delay), [seconds]
   //  TIME_WRN_L_ON_DEL        TIMER — Low warning on delay time          Real
   //                      (activation delay), [seconds]
   //  TIME_ALM_H_OFF_DEL      TIMER — High alarm off delay time           Real
   //                      (deactivation delay), [seconds]
   //  TIME_ALM_L_OFF_DEL       TIMER — Low alarm off delay time            Real
   //                      (deactivation delay), [seconds]
   //  TIME_WRN_H_OFF_DEL      TIMER — High warning off delay time          Real
   //                      (deactivation delay), [seconds]
   //  TIME_WRN_L_OFF_DEL      TIMER — Low warning off delay time           Real
   //                      (deactivation delay), [seconds]
   //  ――――――――――――――――――――――――――――――――――――――――――
   // 
   // 
   // 
   // ▂▂▂▂▂▂▂▂▂▂▂▂▂▂▂▂▂▂▂▂▂▂▂▂▂▂▂▂▂▂▂▂▂▂▂▂▂▂▂▂▂▂▂▂
   // 6.4      UT22001_Dy_InstAnalogRead
   // 
   // 
   // The static data structure for an analog instrument.
   // 
   // 
   //  UT22001_Dy_InstAnalogReadl (full contents)
   //  ――――――――――――――――――――――――――――――――――――――――――
   //  SIGNAL NAME          FUNCTION                     TYPE
   //  ――――――――――――――――――――――――――――――――――――――――――
   //  status_ConfigError       STATUS — Raw or scaled range configuration error   Bool
   //                      (1 = Config error, 0 = OK)
   //  status_Alm_H         STATUS — High alarm is active           Bool
   //                      (1 = alarm active, 0 = no alarm)
   //  status_Alm_L          STATUS — Low alarm is active            Bool
   //                      (1 = alarm active, 0 = no alarm)
   //  status_Wrn_H         STATUS — High warning is active          Bool
   //                      (1 = warning active, 0 = no warning)
   //  status_Wrn_L          STATUS — Low warning is active           Bool
   //                      (1 = warning active, 0 = no warning)
   //  status_Alm_H_Mask       STATUS — High alarm is masked             Bool
   //                      (1 = alarm masked, 0 = normal)
   //  status_Alm_L_Mask        STATUS — Low alarm is masked              Bool
   //                      (1 = alarm masked, 0 = normal)
   //  status_Wrn_H_Mask       STATUS — High warning is masked            Bool
   //                      (1 = warning masked, 0 = normal)
   //  status_Wrn_L_Mask        STATUS — Low warning is masked             Bool
   //                      (1 = warning masked, 0 = normal)
   //  status_Alm_H_Dis           STATUS — High alarm is disabled            Bool
   //                      (1 = alarm disabled, 0 = normal)
   //  status_Alm_L_Dis            STATUS — Low alarm is disabled             Bool
   //                      (1 = alarm disabled, 0 = normal)
   //  status_Wrn_H_Dis           STATUS — High warning is disabled           Bool
   //                      (1 = warning disabled, 0 = normal)
   //  status_Wrn_L_Dis            STATUS — Low warning is disabled            Bool
   //                      (1 = warning disabled, 0 = normal)
   //  status_Fault            STATUS — Instrument is in fault             Bool
   //                      (1 = fault present, 0 = healthy)
   //  status_SimOn           STATUS — Device is in simulation mode             Bool
   //                      (1 = Simulation mode, 0 = normal)
   //  status_RemoteOn       STATUS — Device is in remote mode                  Bool
   //                      (1 = Remote mode, 0 = normal)
   //  status_LocalOn         STATUS — Device is in local mode                 Bool
   //                      (1 = Local mode, 0 = normal)
   //  status_RLOff         STATUS — Device is in ALL mode                   Bool
   //                      (1 = ALL mode, 0 = normal)
   // 
   //  cal_OR_Abs          CALC — Over-range limit (absolute value)      Real
   //  cal_UR_Abs          CALC — Under-range limit (absolute value)       Real
   // 
   //  mode_Alm_H_MaskOn     MODE — Masks the high alarm             Bool    
   //                    (1 = alarm masked, 0 = normal)
   //  mode_Alm_L_MaskOn     MODE — Masks the low alarm            Bool    
   //                    (1 = alarm masked, 0 = normal)
   //  mode_Wrn_H_MaskOn     MODE — Masks the high warning            Bool    
   //                    (1 = warning masked, 0 = normal)
   //  mode_Wrn_L_MaskOn      MODE — Masks the low warning                 Bool    
   //                    (1 = warning masked, 0 = normal)
   //  mode_SimOn         MODE — Simulation mode               Bool
   //                    (1 = sim mode active, 0 = normal)
   //  mode_SimValue       MODE — Simulation value               Real
   //                    (engineering units)
   //  mode_RemoteOn        MODE — Remote SCADA control enabled       Bool
   //                    (1 = active, 0 = disabled or N/A)
   //  mode_LocalOn         MODE — Local HMI control enabled           Bool
   //                    (1 = active, 0 = disabled or N/A)
   // 
   //  msg_Alm_H         MESSAGE — Alarm - high alarm is active        Bool
   //  msg_Alm_L          MESSAGE — Alarm - low alarm is active          Bool
   //  msg_Wrn_H          MESSAGE — Warning - high warning is active      Bool
   //  msg_Wrn_L          MESSAGE — Warning - low warning is active        Bool
   //  msg_Flt_External         MESSAGE — Fault - external fault signal is active      Bool
   //  msg_Flt_OverRange¹     MESSAGE — Fault - instrument is over-range       Bool
   //  msg_Flt_UnderRange¹      MESSAGE — Fault - instrument is under-range       Bool
   //  msg_Flt_OutOfRange¹      MESSAGE — Fault - instrument is out-of-range        Bool
   // 
   //  batch_ID         BATCH — Booking ID (optional for batch operations)   UInt
   // 
   //  actual_Value          ACTUAL — SCALED INSTRUMENT VALUE         Real
   //                      [engineering units]
   //  actual_Alm_H_Timer      ACTUAL — Timer value — alarm high operation     Real
   //                      timer [seconds]
   //  actual_Alm_L_Timer       ACTUAL — Timer value — alarm low operation    Real
   //                      timer [seconds]
   //  actual_Wrn_H_Timer      ACTUAL — Timer value — warning high operation    Real
   //                      timer [seconds]
   //  actual_Wrn_L_Timer       ACTUAL — Timer value — warning low operation      Real
   //                      timer [seconds]
   //  actual_AiRawData       ACTUAL — Analog input Raw Data in use         UT00801
   //                      A copy of the AI_RAW_DATA parameter
   //  actual_AiScaleData     ACTUAL — Analog input Scale Data in use      UT00851
   //                      A copy of the AI_SCALE_DATA parameter
   // 
   //  $pret_AlmHEn           INTERNAL — Edge retention (+ve) alarm high en      Bool
   //  $Pret_AlmLEn            INTERNAL — Edge retention (+ve) alarm low en     Bool
   //  $pret_WrnHEn           INTERNAL — Edge retention (+ve) warning high en     Bool
   //  $pret_WrnLEn            INTERNAL — Edge retention (+ve) warning low en       Bool
   //  ――――――――――――――――――――――――――――――――――――――――――
   //  ¹        msg_Flt_OverRange, msg_Flt_UnderRange and msg_Flt_OutOfRange will all
   //      activate if a configuration error is active status_ConfigError = 1, actual_Value will 
   //      also be set to zero under these conditions.
   // 
   // 
   // With the exception of the flowing, all these signals are discussed in the previous sections, the 
   // outstanding items are firstly:
   // 
   //      batch_ID
   // 
   // The batch_ID is not required for normal use; it is only used where a “booking” system is used 
   // (common in batch and routing applications). Such booking applications can acquire the device 
   // if it is free and reserve it for a particular phase of the batch. Batch applications are a topic in 
   // their own right and are discussed separately in the online User Guide.
   // 
   // Next:
   //      actual_Alm_H_Timer Real
   //      actual_Alm_L_Timer Real
   //      actual_Wrn_H_Timer Real
   //      actual_Wrn_L_Timer Real
   // 
   // These data points hold the actual value of the running timer for each of the alarms/warnings, 
   // both on and off-delay timers used the same timer within the block (the timers are mutually 
   // exclusive, only one will be running at once for each alarm or warning — hence only one timer is
   // needed for each alarm or warning).
   // 
   // Each timer counts down from the TIME_ values (UT02001_St_InstAnalogRead) to zero in 200 ms
   // intervals.
   // 
   // Finally:
   //      $pret_AlmHEn
   //      $Pret_AlmLEn
   //      $pret_WrnHEn
   //      $pret_WrnLEn
   // 
   // These are internal working signals (all signals the start with a $ are internal working signals 
   // used by the block). In this instance they are used to detect a rising edge on each of the alarm 
   // and warning enable signals. 
   // 
   //                ━━━   ⬙⬙⬙⬙⬙⬙   ━━━
   // 
   // 
   // 
   // ▄▄▄▄▄▄▄▄▄▄▄▄▄▄▄▄▄▄▄▄▄▄▄▄▄▄▄▄▄▄▄▄▄▄▄▄▄▄▄▄▄▄▄▄
   // 7.     CONSTANTS AND TEMPORARY (LOCAL) DATA
   // 
   // 
   // 
   // ▂▂▂▂▂▂▂▂▂▂▂▂▂▂▂▂▂▂▂▂▂▂▂▂▂▂▂▂▂▂▂▂▂▂▂▂▂▂▂▂▂▂▂▂
   // 7.1     Constants
   // 
   // 
   // No constants are used in this block.
   // 
   // 
   // 
   // ▂▂▂▂▂▂▂▂▂▂▂▂▂▂▂▂▂▂▂▂▂▂▂▂▂▂▂▂▂▂▂▂▂▂▂▂▂▂▂▂▂▂▂▂
   // 7.2     Temporary (local) data
   // 
   // 
   // The following temporary data is used:
   // 
   // 
   //  Temporary (local) data
   //  ――――――――――――――――――――――――――――――――――――――――――
   //  SIGNAL NAME          FUNCTION                  TYPE
   //  ――――――――――――――――――――――――――――――――――――――――――
   //  revInfo             Revision information for the block         UT01000
   //  licInfo           Licensing information for the block      UT01001
   //  wrkAlmHEn          Working Alm_H is enabled and not masked   Bool
   //  wrkAlmLEn        Working Alm_L is enabled and not masked    Bool
   //  wrkWrnHEn           Working Wrn_H is enabled and not masked    Bool
   //  wrkWrnLEn           Working Wrn_L is enabled and not masked    Bool
   //  calPart1             Scale value part 1 (AI_RAW_SIGNAL − RAW_MIN)Real
   //  calPart2             Scale value part 2 (SCALE_MAX − SCALE_MIN)   Real
   //  calPart3             Scale value part 3 (RAW_MAX − RAW_MIN)     Real
   //  calAbsOOR           Calculated OOR absolute value          Real
   //  calHystAbs           Absolute hysteresis value           Real
   //  wrkHyst           Working hysteresis value            Real
   //  wrkOORPercent         Working out of range percentage          Real
   //  wrkInt           Working storage area (integer)          Int
   //  wrkReal           Working storage (Real)             Real
   //  wrkDInt           Working storage area (double integer)         DInt
   //  ――――――――――――――――――――――――――――――――――――――――――
   // 
   //                ━━━   ⬙⬙⬙⬙⬙⬙   ━━━
   // 
   // 
   // 
   // ▄▄▄▄▄▄▄▄▄▄▄▄▄▄▄▄▄▄▄▄▄▄▄▄▄▄▄▄▄▄▄▄▄▄▄▄▄▄▄▄▄▄▄▄
   // 8.     BLOCK CALLS AND ASSOCIATIONS
   // 
   // 
   // This section details any blocks which may be called from within this software module (subroutine 
   // functions for example), any partner blocks with which it may be associated (for example a 
   // receive module that is partner with a transmit module &c.). It lists any system functions which 
   // may be called (e.g. reading the real time clock) and any system data types that may be used.
   // 
   // Finally, it lists any special calling requirements for the block (for example, must be called from 
   // within a cyclic interrupt organisation block) and if the block is using “optimised access” (this is 
   // the default arrangement).
   // 
   // 
   // 
   // ▂▂▂▂▂▂▂▂▂▂▂▂▂▂▂▂▂▂▂▂▂▂▂▂▂▂▂▂▂▂▂▂▂▂▂▂▂▂▂▂▂▂▂▂
   // 8.1     Block calls from within this module
   // 
   // 
   // There are no PAL block calls from within this block.
   // 
   // 
   // 
   // ▂▂▂▂▂▂▂▂▂▂▂▂▂▂▂▂▂▂▂▂▂▂▂▂▂▂▂▂▂▂▂▂▂▂▂▂▂▂▂▂▂▂▂▂
   // 8.2     Blocks associated with this module
   // 
   // 
   // This is a stand-alone block and is not associated with any other blocks.
   // 
   // 
   // 
   // ▂▂▂▂▂▂▂▂▂▂▂▂▂▂▂▂▂▂▂▂▂▂▂▂▂▂▂▂▂▂▂▂▂▂▂▂▂▂▂▂▂▂▂▂
   // 8.3     System block calls and system data types
   // 
   // There are no system block calls
   // 
   // 
   // 
   // ▂▂▂▂▂▂▂▂▂▂▂▂▂▂▂▂▂▂▂▂▂▂▂▂▂▂▂▂▂▂▂▂▂▂▂▂▂▂▂▂▂▂▂▂
   // 8.4     Special properties and requirements
   // 
   // 
   // 
   // ▁▁▁▁▁▁▁▁▁▁▁▁▁▁▁▁▁▁▁▁▁▁▁▁▁▁▁▁▁▁▁▁▁▁▁▁▁▁▁▁▁▁▁▁
   // 8.4.1     Block optimisation, IEC compatibility and library conformance
   // 
   // 
   //    •   Block optimisation is ACTIVE for this block.
   // 
   //    •   The block has been checked for IEC compatibility and is compliant.
   // 
   //    •   The block is compatible with all IEC library-conformance module constraints
   // 
   // 
   // 
   // ▁▁▁▁▁▁▁▁▁▁▁▁▁▁▁▁▁▁▁▁▁▁▁▁▁▁▁▁▁▁▁▁▁▁▁▁▁▁▁▁▁▁▁▁
   // 8.4.2     Calling requirements
   // 
   // 
   // There are no special calling requirements for this block.
   // 
   //                ━━━   ⬙⬙⬙⬙⬙⬙   ━━━
   // 
   // 
   // 
   // ▄▄▄▄▄▄▄▄▄▄▄▄▄▄▄▄▄▄▄▄▄▄▄▄▄▄▄▄▄▄▄▄▄▄▄▄▄▄▄▄▄▄▄▄
   // 9.     EXAMPLE USAGE
   // 
   // 
   // The following shows a typical deployment of FC02001:
   // 
   // 
   //                            ┌─────────────
   //         ───────────────────┤ FC02001 
   //                            │               │                       
   //                                "FC001" ─┤ AI_RAW_SIGNAL          │
   //                            │               │
   //       "DB00801_St_ConstAiRawData".AI_RAW_2003 ─┤ AI_RAW_DATA           │
   //                            │               │
   //    "DB00851_St_ConstAiScaleData".AI_SCALE_FC001    ─┤ AI_SCALE_DATA          │
   //                            │               │
   //              "FC001_FAULT"           │               │
   //           ────┤╱├──────────┤ EXT_FAULT                │
   //                            │               │
   //                            │               │
   //         "DB02001_St_StdInstAnalogRead".FC001 ─┤ STATIC_DATA             │
   //                            │
   //        "DB22001_Dy_StdInstAnalogRead".FC001 ─┤ DYNAMIC_DATA
   //                            │
   //                            │
   // 
   // 
   //               ━━━   ⬙⬙⬙⬙⬙⬙   ━━━
   // 
   // 
   // 
   // ▄▄▄▄▄▄▄▄▄▄▄▄▄▄▄▄▄▄▄▄▄▄▄▄▄▄▄▄▄▄▄▄▄▄▄▄▄▄▄▄▄▄▄▄
   // 10.     TEST AND VERIFICATION PATH
   // 
   // 
   // The following diagram shows the full test and verification path for the formal release of each 
   // version of the software module. See the Test Plan [Ref. 003] for full details, available here:
   //         https://psop.uk/pal-tp-p
   // 
   // 
   //         FC02001-T001         FC02001-T002         FC02001-T003
   // 
   //     Test version: 000.801     Test version: 001.801     Test version: 002.801
   //  Released version: 001.000     Released version: 002.000     Released version: 003.000
   // Released commit: D0008    Released commit: D0011    Released commit: D0018
   // 
   //        SCR      SMT         SCR      SMT                 SMTp  
   // ＿＿＿＿＿＿┌┐＿＿ ▛▜ ＿＿＿＿＿＿＿＿┌┐＿＿ ▛▜ ＿＿＿＿＿＿＿＿＿＿＿＿ ▛ ┐＿＿
   //       └┘   ▙▟         └┘   ▙▟             └ ▟   
   // Initial test           IEC compliance       AI_RAW_DATA & AI_SCALE_DATA
   // 
   // Initial test to release the      Comments updated &    DB00801 and DB00851 added 
   // module following the      UDT  variable names       and used throughout, minor 
   // development stage.       standardised        name changes, comments 
   // Full SMT              Full SMT            updated. Only a partial retest 
   //                             required
   // 
   // Where:
   // ――――――――――――――――――――――――――――――――――――――――――――
   //  SCR    Source Code Review      A visual inspection of the software to ensure it has been written  
   // ┌┐             to the correct standards, uses the correct structures within the
   // └┘             software and is generally suitable for deployment.               
   // 
   //  SMT Software Module Test    A full and detailed test of an individual software module in
   //   ▛▜              isolation; such testing requires that all branches of the 
   //   ▙▟              software are tested. 
   // 
   //                It tests all the interfaces to the module, any data recorded or 
   //                stored by the module, all error and exception handling functions 
   //                and tests all timed and interrupt driven operations.
   // 
   //  SMTp SMT partial retest      A partial repeat of some aspect of the full SMT to retest a small
   //   ▛ ┐               change made to some aspect of the software. The change 
   // └ ▟                must be small, specific and localised.
   // 
   //  SCV Software Compatibility     A mechanism for verifying that no executable code software 
   // ╓╖    Verification          changes have been made to a module following changes to
   // ╙╜             comment fields.
   // 
   //                Allows typographical errors &c. to be corrected without forcing 
   //                a full SMT on a module that has not functionally changed.
   // ――――――――――――――――――――――――――――――――――――――――――――
   // 
   // An SCV can only be performed on a module that has at some point previously, successfully 
   // completed both an SCR and SMT. Where an SCV is implemented, it replaces the requirement for 
   // both the SCR and the SMT for the test iteration in question.
   // 
   //                ━━━   ⬙⬙⬙⬙⬙⬙   ━━━
   // 
   // 
   // 
   // ██████████████ █ █ █ █  END   █ █ █ █ ██████████████
END_REGION

REGION Network 4: Current revision and modification history
   // ▄▄▄▄▄▄▄▄▄▄▄▄▄▄▄▄▄▄▄▄▄▄▄▄▄▄▄▄▄▄▄▄▄▄▄▄▄▄▄▄▄▄▄▄
   // MODIFICATION HISTORY
   // 
   // 
   // The revision data shown here, in the network comments, contains additional information 
   // reflecting the software development workflow under the version control system (VCS) employed 
   // to track all software changes.
   // 
   // The VCS in use is the Git Source Code Management system in conjunction with the GitHub online 
   // hosting system. The software in its entirety is available in the GitHub remote repository:
   // 
   //      https://github.com/practicalseries/PS2001-pal-software
   // 
   // The repository is public and can be freely copied (forked in GitHub terminology) and used 
   // under the MIT licence. 
   // 
   // The MIT licence is reproduced in full in the last network of this software module.
   // 
   // 
   //  ―――――――――――――――――――――――――――――――――――――――――――
   //  DATE       REVISION             MASTER BRANCH     DEV
   //          (nnn.amm)   COMMIT TAG    (Base ---> Merge)    BRANCH   Author
   //  ———————————————————————————————————————————
   //  2024.05.11    002.801   D0017A-000.104   D0017 N/A     D017A   M. Gledhill
   //                        RAW_ANALOG changed to AI_RAW_SIGNAL
   //                        AI_RAW_DATA and AI_SCALE_DATA added and
   //                        copied to DYNAMIC_DATA (see db00801 SMDS)
   // 
   //  2022.04.16    002.000   D0011      D0010 D0011  None  M. Gledhill
   //                        FC02001 — RELEASED FOR USE
   //                          Merge back to master branch
   // 
   //  2022.04.11    001.801   D0010A-000.801   D0010 N/A     D010A   M. Gledhill
   //                        Released for test (SCV)
   //  2022.04.08    001.102   D0010A-000.104   D0010 N/A     D010A   M. Gledhill
   //                        Temporary variable name change (cal)
   // 
   //  2022.04.05    001.101   D0010A-000.103   D0010 N/A     D010A   M. Gledhill
   //                        Over and under range based on scaled signal
   //                        INFO_TYPE, cal_OR_Abs and cal_UR_Abs added
   //                        Comments updated and standardised
   //                        UDT variable names standardised
   // 
   //  2021.05.26    001.000   D0008      D0006 D0008  None    M. Gledhill
   //                        FC02001 — RELEASED FOR USE
   //                          Merge back to master branch
   // 
   //  2021.05.26    001.000   D0006B-001.000   D0006 N/A     D0006B   M. Gledhill
   //                        FC02001 — Post-test RELEASED FOR USE
   // 
   //  2021.05.24    000.801   D0006B-000.801   D0006 N/A     D0006B   M. Gledhill
   //                        FC02001 — Released for SMT
   // 
   //  2021.05.18    000.101   D0006B-000.101   D0006 N/A     D0006B   M. Gledhill
   //                        FC02001 Migration to VCS
   //  ———————————————————————————————————————————
   //   Where: nnn  =  Major revision
   //         a  =  Type (1-7 Development, 8 Proving, 9 Qualification, 0 Release)
   //       mm  =  Minor revision (must be 00 if a = 0)
   //         Block properties version number should be set to nn.a (only one decimal place)
   // 
   // ▄▄▄▄▄▄▄▄▄▄▄▄▄▄▄▄▄▄▄▄▄▄▄▄▄▄▄▄▄▄▄▄▄▄▄▄▄▄▄▄▄▄▄▄
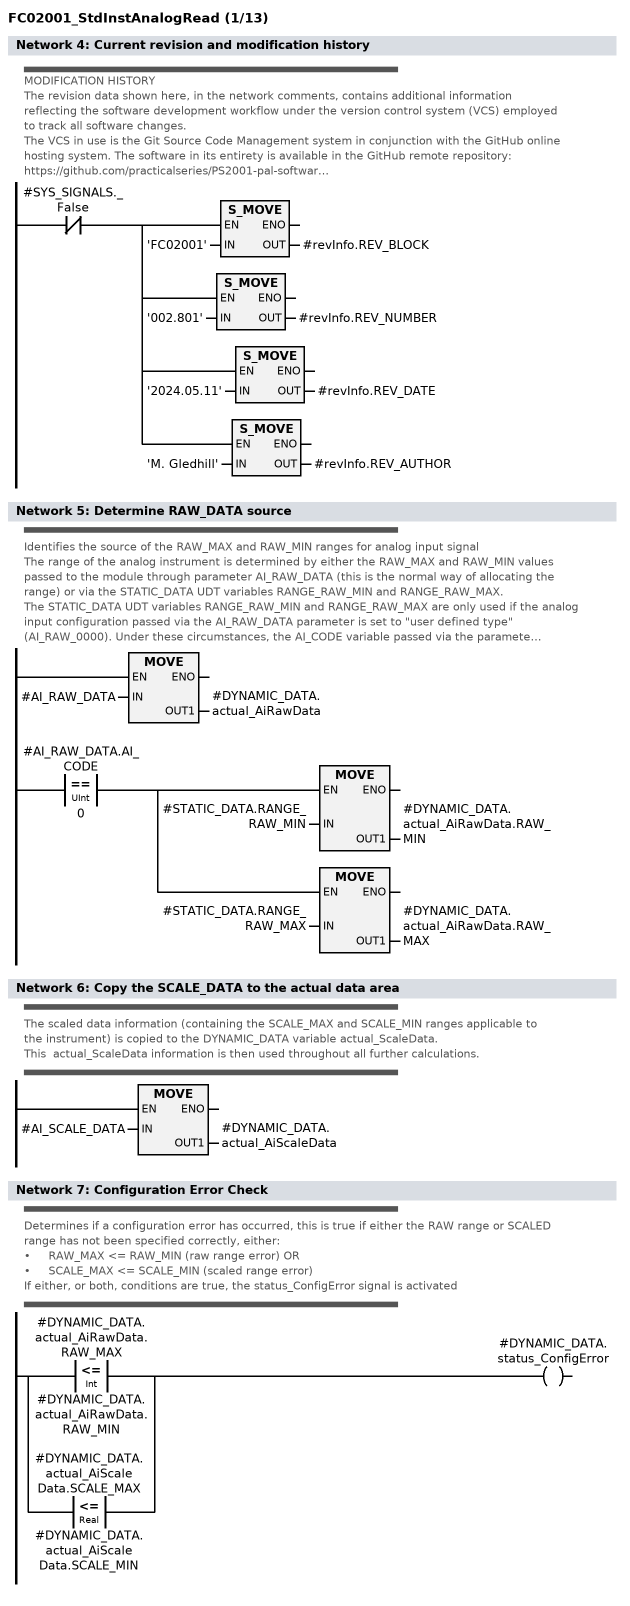
   RUNG wire#powerrail
      I_Contact( #SYS_SIGNALS._False )
      wire#w1
      S_Move(in := 'FC02001', out => #revInfo.REV_BLOCK)
   END_RUNG
   RUNG wire#w1
      S_Move(in := '002.801', out => #revInfo.REV_NUMBER)
   END_RUNG
   RUNG wire#w1
      S_Move(in := '2024.05.11', out => #revInfo.REV_DATE)
   END_RUNG
   RUNG wire#w1
      S_Move(in := 'M. Gledhill', out => #revInfo.REV_AUTHOR)
   END_RUNG
   // the same network as SCL:
   IF NOT #SYS_SIGNALS._False THEN
       #revInfo.REV_BLOCK := 'FC02001';
       #revInfo.REV_NUMBER := '002.801';
       #revInfo.REV_DATE := '2024.05.11';
       #revInfo.REV_AUTHOR := 'M. Gledhill';
   END_IF;
END_REGION

REGION Network 5: Determine RAW_DATA source
   // ▀▀▀▀▀▀▀▀▀▀▀▀▀▀▀▀▀▀▀▀▀▀▀▀▀▀▀▀▀▀▀▀▀▀▀▀▀▀▀▀▀▀▀▀
   // Identifies the source of the RAW_MAX and RAW_MIN ranges for analog input signal
   // 
   // The range of the analog instrument is determined by either the RAW_MAX and RAW_MIN values 
   // passed to the module through parameter AI_RAW_DATA (this is the normal way of allocating the 
   // range) or via the STATIC_DATA UDT variables RANGE_RAW_MIN and RANGE_RAW_MAX.
   // 
   // 
   // The STATIC_DATA UDT variables RANGE_RAW_MIN and RANGE_RAW_MAX are only used if the analog
   // input configuration passed via the AI_RAW_DATA parameter is set to "user defined type" 
   // (AI_RAW_0000). Under these circumstances, the AI_CODE variable passed via the parameter 
   // AI_RAW_DATA will be set to zero and the STATIC_DATA UDT variables RANGE_RAW_MIN and 
   // RANGE_RAW_MAX are to be used in place of the range data given via the AI_RAW_DATA parameter.
   // 
   // Irrespective of the source, the RAW_MIN and RAW_MAX data in use will be copied to the 
   // DYNAMIC_DATA variable actual_RawData.
   // ▄▄▄▄▄▄▄▄▄▄▄▄▄▄▄▄▄▄▄▄▄▄▄▄▄▄▄▄▄▄▄▄▄▄▄▄▄▄▄▄▄▄▄▄
   RUNG wire#powerrail
      Move(in := #AI_RAW_DATA, out1 => #DYNAMIC_DATA.actual_AiRawData)
   END_RUNG
   RUNG wire#powerrail
      { S7_Templates := "SrcType := UInt" } EQ_Contact(in1 := #AI_RAW_DATA.AI_CODE, in2 := 0)
      wire#w1
      Move(in := #STATIC_DATA.RANGE_RAW_MIN, out1 => #DYNAMIC_DATA.actual_AiRawData.RAW_MIN)
   END_RUNG
   RUNG wire#w1
      Move(in := #STATIC_DATA.RANGE_RAW_MAX, out1 => #DYNAMIC_DATA.actual_AiRawData.RAW_MAX)
   END_RUNG
   // the same network as SCL:
   #DYNAMIC_DATA.actual_AiRawData := #AI_RAW_DATA;
   IF #AI_RAW_DATA.AI_CODE = 0 THEN
       #DYNAMIC_DATA.actual_AiRawData.RAW_MIN := #STATIC_DATA.RANGE_RAW_MIN;
       #DYNAMIC_DATA.actual_AiRawData.RAW_MAX := #STATIC_DATA.RANGE_RAW_MAX;
   END_IF;
END_REGION

REGION Network 6: Copy the SCALE_DATA to the actual data area
   // ▀▀▀▀▀▀▀▀▀▀▀▀▀▀▀▀▀▀▀▀▀▀▀▀▀▀▀▀▀▀▀▀▀▀▀▀▀▀▀▀▀▀▀▀
   // The scaled data information (containing the SCALE_MAX and SCALE_MIN ranges applicable to
   // the instrument) is copied to the DYNAMIC_DATA variable actual_ScaleData.
   // 
   // This  actual_ScaleData information is then used throughout all further calculations.
   // ▄▄▄▄▄▄▄▄▄▄▄▄▄▄▄▄▄▄▄▄▄▄▄▄▄▄▄▄▄▄▄▄▄▄▄▄▄▄▄▄▄▄▄▄
   RUNG wire#powerrail
      Move(in := #AI_SCALE_DATA, out1 => #DYNAMIC_DATA.actual_AiScaleData)
   END_RUNG
   // the same network as SCL:
   #DYNAMIC_DATA.actual_AiScaleData := #AI_SCALE_DATA;
END_REGION

REGION Network 7: Configuration Error Check
   // ▀▀▀▀▀▀▀▀▀▀▀▀▀▀▀▀▀▀▀▀▀▀▀▀▀▀▀▀▀▀▀▀▀▀▀▀▀▀▀▀▀▀▀▀
   // Determines if a configuration error has occurred, this is true if either the RAW range or SCALED 
   // range has not been specified correctly, either:
   // 
   //    •   RAW_MAX <= RAW_MIN (raw range error) OR
   //    •   SCALE_MAX <= SCALE_MIN (scaled range error)
   // 
   // If either, or both, conditions are true, the status_ConfigError signal is activated
   // ▄▄▄▄▄▄▄▄▄▄▄▄▄▄▄▄▄▄▄▄▄▄▄▄▄▄▄▄▄▄▄▄▄▄▄▄▄▄▄▄▄▄▄▄
   RUNG wire#powerrail
      { S7_Templates := "SrcType := Int" } LE_Contact(in1 := #DYNAMIC_DATA.actual_AiRawData.RAW_MAX, in2 := #DYNAMIC_DATA.actual_AiRawData.RAW_MIN)
      wire#w1
      Coil( #DYNAMIC_DATA.status_ConfigError )
   END_RUNG
   RUNG wire#powerrail
      { S7_Templates := "SrcType := Real" } LE_Contact(in1 := #DYNAMIC_DATA.actual_AiScaleData.SCALE_MAX, in2 := #DYNAMIC_DATA.actual_AiScaleData.SCALE_MIN)
   END_RUNG wire#w1
   // the same network as SCL:
   #DYNAMIC_DATA.status_ConfigError := (#DYNAMIC_DATA.actual_AiRawData.RAW_MAX <= #DYNAMIC_DATA.actual_AiRawData.RAW_MIN) OR (#DYNAMIC_DATA.actual_AiScaleData.SCALE_MAX <= #DYNAMIC_DATA.actual_AiScaleData.SCALE_MIN);
END_REGION

REGION Network 8: Signal Conditioning — Simulation mode disabled
   // ▀▀▀▀▀▀▀▀▀▀▀▀▀▀▀▀▀▀▀▀▀▀▀▀▀▀▀▀▀▀▀▀▀▀▀▀▀▀▀▀▀▀▀▀
   // If simulation mode is disabled (CONFIG_SIM_DIS = 1), or if the faceplate is disabled 
   // (CONFIG_FP_DIS = 1),reset any simulation mode activation signal.
   // ▄▄▄▄▄▄▄▄▄▄▄▄▄▄▄▄▄▄▄▄▄▄▄▄▄▄▄▄▄▄▄▄▄▄▄▄▄▄▄▄▄▄▄▄
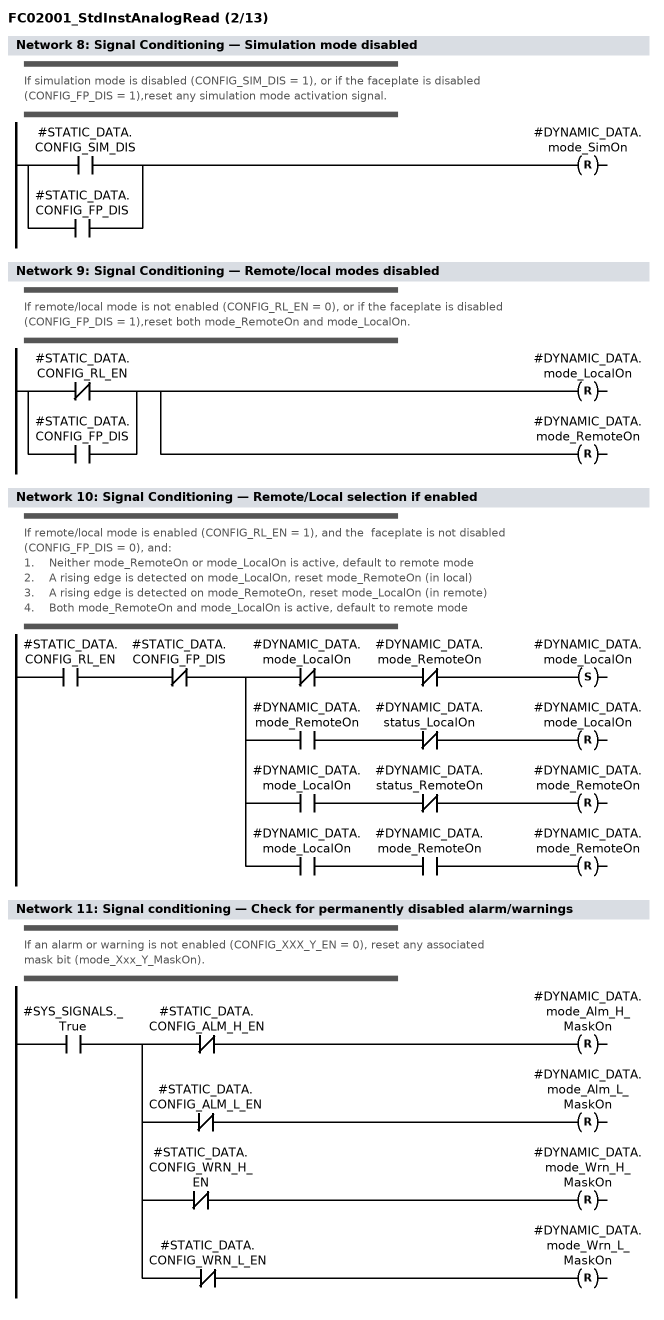
   RUNG wire#powerrail
      Contact( #STATIC_DATA.CONFIG_SIM_DIS )
      wire#w1
      R_Coil( #DYNAMIC_DATA.mode_SimOn )
   END_RUNG
   RUNG wire#powerrail
      Contact( #STATIC_DATA.CONFIG_FP_DIS )
   END_RUNG wire#w1
   // the same network as SCL:
   IF #STATIC_DATA.CONFIG_SIM_DIS OR #STATIC_DATA.CONFIG_FP_DIS THEN
       #DYNAMIC_DATA.mode_SimOn := FALSE;
   END_IF;
END_REGION

REGION Network 9: Signal Conditioning — Remote/local modes disabled
   // ▀▀▀▀▀▀▀▀▀▀▀▀▀▀▀▀▀▀▀▀▀▀▀▀▀▀▀▀▀▀▀▀▀▀▀▀▀▀▀▀▀▀▀▀
   // If remote/local mode is not enabled (CONFIG_RL_EN = 0), or if the faceplate is disabled 
   // (CONFIG_FP_DIS = 1),reset both mode_RemoteOn and mode_LocalOn.
   // ▄▄▄▄▄▄▄▄▄▄▄▄▄▄▄▄▄▄▄▄▄▄▄▄▄▄▄▄▄▄▄▄▄▄▄▄▄▄▄▄▄▄▄▄
   RUNG wire#powerrail
      I_Contact( #STATIC_DATA.CONFIG_RL_EN )
      wire#w1
      R_Coil( #DYNAMIC_DATA.mode_LocalOn )
   END_RUNG
   RUNG wire#powerrail
      Contact( #STATIC_DATA.CONFIG_FP_DIS )
   END_RUNG wire#w1
   RUNG wire#w1
      R_Coil( #DYNAMIC_DATA.mode_RemoteOn )
   END_RUNG
   // the same network as SCL:
   IF NOT #STATIC_DATA.CONFIG_RL_EN OR #STATIC_DATA.CONFIG_FP_DIS THEN
       #DYNAMIC_DATA.mode_LocalOn := FALSE;
       #DYNAMIC_DATA.mode_RemoteOn := FALSE;
   END_IF;
END_REGION

REGION Network 10: Signal Conditioning — Remote/Local selection if enabled
   // ▀▀▀▀▀▀▀▀▀▀▀▀▀▀▀▀▀▀▀▀▀▀▀▀▀▀▀▀▀▀▀▀▀▀▀▀▀▀▀▀▀▀▀▀
   // If remote/local mode is enabled (CONFIG_RL_EN = 1), and the  faceplate is not disabled 
   // (CONFIG_FP_DIS = 0), and:
   // 
   //    1.  Neither mode_RemoteOn or mode_LocalOn is active, default to remote mode
   //    2.  A rising edge is detected on mode_LocalOn, reset mode_RemoteOn (in local)
   //    3.  A rising edge is detected on mode_RemoteOn, reset mode_LocalOn (in remote)
   //    4.  Both mode_RemoteOn and mode_LocalOn is active, default to remote mode
   // ▄▄▄▄▄▄▄▄▄▄▄▄▄▄▄▄▄▄▄▄▄▄▄▄▄▄▄▄▄▄▄▄▄▄▄▄▄▄▄▄▄▄▄▄
   RUNG wire#powerrail
      Contact( #STATIC_DATA.CONFIG_RL_EN )
      I_Contact( #STATIC_DATA.CONFIG_FP_DIS )
      wire#w1
      I_Contact( #DYNAMIC_DATA.mode_LocalOn )
      I_Contact( #DYNAMIC_DATA.mode_RemoteOn )
      S_Coil( #DYNAMIC_DATA.mode_LocalOn )
   END_RUNG
   RUNG wire#w1
      Contact( #DYNAMIC_DATA.mode_RemoteOn )
      I_Contact( #DYNAMIC_DATA.status_LocalOn )
      R_Coil( #DYNAMIC_DATA.mode_LocalOn )
   END_RUNG
   RUNG wire#w1
      Contact( #DYNAMIC_DATA.mode_LocalOn )
      I_Contact( #DYNAMIC_DATA.status_RemoteOn )
      R_Coil( #DYNAMIC_DATA.mode_RemoteOn )
   END_RUNG
   RUNG wire#w1
      Contact( #DYNAMIC_DATA.mode_LocalOn )
      Contact( #DYNAMIC_DATA.mode_RemoteOn )
      R_Coil( #DYNAMIC_DATA.mode_RemoteOn )
   END_RUNG
   // the same network as SCL:
   #_w1 := #STATIC_DATA.CONFIG_RL_EN AND NOT #STATIC_DATA.CONFIG_FP_DIS;
   IF #_w1 AND NOT #DYNAMIC_DATA.mode_LocalOn AND NOT #DYNAMIC_DATA.mode_RemoteOn THEN
       #DYNAMIC_DATA.mode_LocalOn := TRUE;
   END_IF;
   IF #_w1 AND #DYNAMIC_DATA.mode_RemoteOn AND NOT #DYNAMIC_DATA.status_LocalOn THEN
       #DYNAMIC_DATA.mode_LocalOn := FALSE;
   END_IF;
   IF #_w1 AND #DYNAMIC_DATA.mode_LocalOn AND NOT #DYNAMIC_DATA.status_RemoteOn THEN
       #DYNAMIC_DATA.mode_RemoteOn := FALSE;
   END_IF;
   IF #_w1 AND #DYNAMIC_DATA.mode_LocalOn AND #DYNAMIC_DATA.mode_RemoteOn THEN
       #DYNAMIC_DATA.mode_RemoteOn := FALSE;
   END_IF;
END_REGION

REGION Network 11: Signal conditioning — Check for permanently disabled alarm/warnings
   // ▀▀▀▀▀▀▀▀▀▀▀▀▀▀▀▀▀▀▀▀▀▀▀▀▀▀▀▀▀▀▀▀▀▀▀▀▀▀▀▀▀▀▀▀
   // If an alarm or warning is not enabled (CONFIG_XXX_Y_EN = 0), reset any associated 
   // mask bit (mode_Xxx_Y_MaskOn).
   // ▄▄▄▄▄▄▄▄▄▄▄▄▄▄▄▄▄▄▄▄▄▄▄▄▄▄▄▄▄▄▄▄▄▄▄▄▄▄▄▄▄▄▄▄
   RUNG wire#powerrail
      Contact( #SYS_SIGNALS._True )
      wire#w1
      I_Contact( #STATIC_DATA.CONFIG_ALM_H_EN )
      R_Coil( #DYNAMIC_DATA.mode_Alm_H_MaskOn )
   END_RUNG
   RUNG wire#w1
      I_Contact( #STATIC_DATA.CONFIG_ALM_L_EN )
      R_Coil( #DYNAMIC_DATA.mode_Alm_L_MaskOn )
   END_RUNG
   RUNG wire#w1
      I_Contact( #STATIC_DATA.CONFIG_WRN_H_EN )
      R_Coil( #DYNAMIC_DATA.mode_Wrn_H_MaskOn )
   END_RUNG
   RUNG wire#w1
      I_Contact( #STATIC_DATA.CONFIG_WRN_L_EN )
      R_Coil( #DYNAMIC_DATA.mode_Wrn_L_MaskOn )
   END_RUNG
   // the same network as SCL:
   IF #SYS_SIGNALS._True AND NOT #STATIC_DATA.CONFIG_ALM_H_EN THEN
       #DYNAMIC_DATA.mode_Alm_H_MaskOn := FALSE;
   END_IF;
   IF #SYS_SIGNALS._True AND NOT #STATIC_DATA.CONFIG_ALM_L_EN THEN
       #DYNAMIC_DATA.mode_Alm_L_MaskOn := FALSE;
   END_IF;
   IF #SYS_SIGNALS._True AND NOT #STATIC_DATA.CONFIG_WRN_H_EN THEN
       #DYNAMIC_DATA.mode_Wrn_H_MaskOn := FALSE;
   END_IF;
   IF #SYS_SIGNALS._True AND NOT #STATIC_DATA.CONFIG_WRN_L_EN THEN
       #DYNAMIC_DATA.mode_Wrn_L_MaskOn := FALSE;
   END_IF;
END_REGION

REGION Network 12: Signal conditioning — Identify alarm/warnings that are to be evaluated
   // ▀▀▀▀▀▀▀▀▀▀▀▀▀▀▀▀▀▀▀▀▀▀▀▀▀▀▀▀▀▀▀▀▀▀▀▀▀▀▀▀▀▀▀▀
   // If an alarm or warning is both ENABLED and NOT MASKED then the associated (local data) 
   // working bit wrkXxxYEn bit is set; this is used in the following networks to indicate that the 
   // alarm/warning is to be evaluated.
   // ▄▄▄▄▄▄▄▄▄▄▄▄▄▄▄▄▄▄▄▄▄▄▄▄▄▄▄▄▄▄▄▄▄▄▄▄▄▄▄▄▄▄▄▄
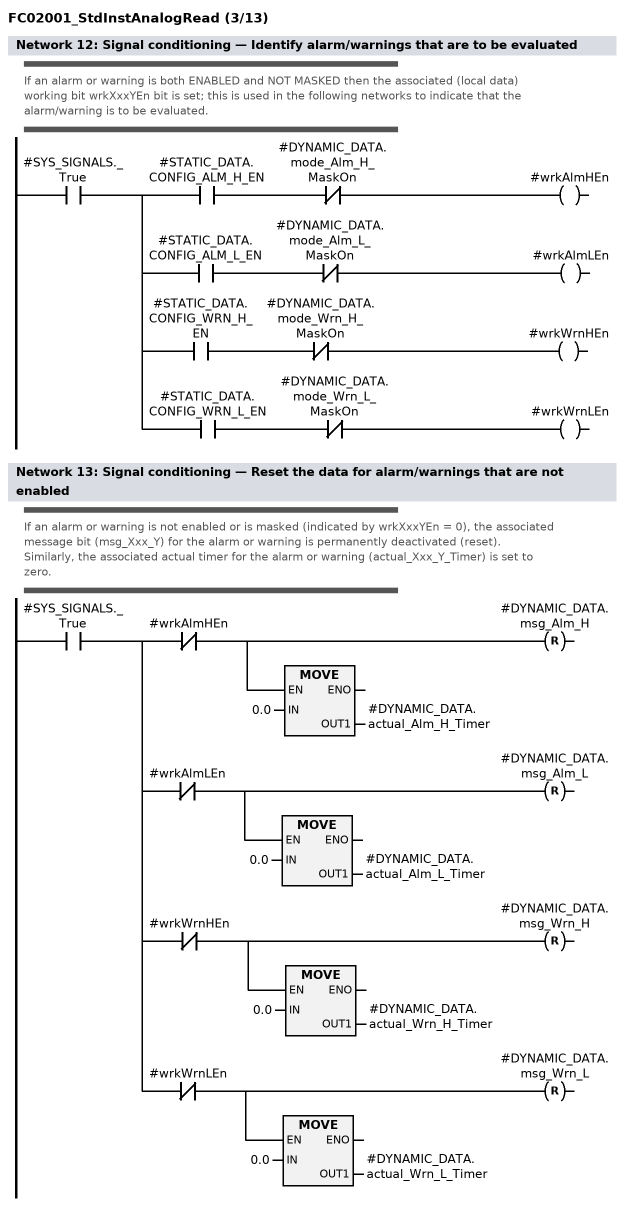
   RUNG wire#powerrail
      Contact( #SYS_SIGNALS._True )
      wire#w1
      Contact( #STATIC_DATA.CONFIG_ALM_H_EN )
      I_Contact( #DYNAMIC_DATA.mode_Alm_H_MaskOn )
      Coil( #wrkAlmHEn )
   END_RUNG
   RUNG wire#w1
      Contact( #STATIC_DATA.CONFIG_ALM_L_EN )
      I_Contact( #DYNAMIC_DATA.mode_Alm_L_MaskOn )
      Coil( #wrkAlmLEn )
   END_RUNG
   RUNG wire#w1
      Contact( #STATIC_DATA.CONFIG_WRN_H_EN )
      I_Contact( #DYNAMIC_DATA.mode_Wrn_H_MaskOn )
      Coil( #wrkWrnHEn )
   END_RUNG
   RUNG wire#w1
      Contact( #STATIC_DATA.CONFIG_WRN_L_EN )
      I_Contact( #DYNAMIC_DATA.mode_Wrn_L_MaskOn )
      Coil( #wrkWrnLEn )
   END_RUNG
   // the same network as SCL:
   #wrkAlmHEn := #SYS_SIGNALS._True AND #STATIC_DATA.CONFIG_ALM_H_EN AND NOT #DYNAMIC_DATA.mode_Alm_H_MaskOn;
   #wrkAlmLEn := #SYS_SIGNALS._True AND #STATIC_DATA.CONFIG_ALM_L_EN AND NOT #DYNAMIC_DATA.mode_Alm_L_MaskOn;
   #wrkWrnHEn := #SYS_SIGNALS._True AND #STATIC_DATA.CONFIG_WRN_H_EN AND NOT #DYNAMIC_DATA.mode_Wrn_H_MaskOn;
   #wrkWrnLEn := #SYS_SIGNALS._True AND #STATIC_DATA.CONFIG_WRN_L_EN AND NOT #DYNAMIC_DATA.mode_Wrn_L_MaskOn;
END_REGION

REGION Network 13: Signal conditioning — Reset the data for alarm/warnings that are not enabled
   // ▀▀▀▀▀▀▀▀▀▀▀▀▀▀▀▀▀▀▀▀▀▀▀▀▀▀▀▀▀▀▀▀▀▀▀▀▀▀▀▀▀▀▀▀
   // If an alarm or warning is not enabled or is masked (indicated by wrkXxxYEn = 0), the associated 
   // message bit (msg_Xxx_Y) for the alarm or warning is permanently deactivated (reset).
   // 
   // Similarly, the associated actual timer for the alarm or warning (actual_Xxx_Y_Timer) is set to 
   // zero.
   // ▄▄▄▄▄▄▄▄▄▄▄▄▄▄▄▄▄▄▄▄▄▄▄▄▄▄▄▄▄▄▄▄▄▄▄▄▄▄▄▄▄▄▄▄
   RUNG wire#powerrail
      Contact( #SYS_SIGNALS._True )
      wire#w1
      I_Contact( #wrkAlmHEn )
      wire#w2
      R_Coil( #DYNAMIC_DATA.msg_Alm_H )
   END_RUNG
   RUNG wire#w2
      { S7_GenerateENO := "TRUE" } Move(in := 0.0, out1 => #DYNAMIC_DATA.actual_Alm_H_Timer)
   END_RUNG
   RUNG wire#w1
      I_Contact( #wrkAlmLEn )
      wire#w3
      R_Coil( #DYNAMIC_DATA.msg_Alm_L )
   END_RUNG
   RUNG wire#w3
      { S7_GenerateENO := "TRUE" } Move(in := 0.0, out1 => #DYNAMIC_DATA.actual_Alm_L_Timer)
   END_RUNG
   RUNG wire#w1
      I_Contact( #wrkWrnHEn )
      wire#w4
      R_Coil( #DYNAMIC_DATA.msg_Wrn_H )
   END_RUNG
   RUNG wire#w4
      { S7_GenerateENO := "TRUE" } Move(in := 0.0, out1 => #DYNAMIC_DATA.actual_Wrn_H_Timer)
   END_RUNG
   RUNG wire#w1
      I_Contact( #wrkWrnLEn )
      wire#w5
      R_Coil( #DYNAMIC_DATA.msg_Wrn_L )
   END_RUNG
   RUNG wire#w5
      { S7_GenerateENO := "TRUE" } Move(in := 0.0, out1 => #DYNAMIC_DATA.actual_Wrn_L_Timer)
   END_RUNG
   // the same network as SCL:
   IF #SYS_SIGNALS._True AND NOT #wrkAlmHEn THEN
       #DYNAMIC_DATA.msg_Alm_H := FALSE;
       #DYNAMIC_DATA.actual_Alm_H_Timer := 0.0;
   END_IF;
   IF #SYS_SIGNALS._True AND NOT #wrkAlmLEn THEN
       #DYNAMIC_DATA.msg_Alm_L := FALSE;
       #DYNAMIC_DATA.actual_Alm_L_Timer := 0.0;
   END_IF;
   IF #SYS_SIGNALS._True AND NOT #wrkWrnHEn THEN
       #DYNAMIC_DATA.msg_Wrn_H := FALSE;
       #DYNAMIC_DATA.actual_Wrn_H_Timer := 0.0;
   END_IF;
   IF #SYS_SIGNALS._True AND NOT #wrkWrnLEn THEN
       #DYNAMIC_DATA.msg_Wrn_L := FALSE;
       #DYNAMIC_DATA.actual_Wrn_L_Timer := 0.0;
   END_IF;
END_REGION

REGION Network 14: Signal conditioning — Detect recently enabled alarm/warnings
   // ▀▀▀▀▀▀▀▀▀▀▀▀▀▀▀▀▀▀▀▀▀▀▀▀▀▀▀▀▀▀▀▀▀▀▀▀▀▀▀▀▀▀▀▀
   // If the working alarm or warning enable signal (wrkXxxYEn) changes to a high state
   // (i.e. the alarm is enabled during run-time), the alarm/warning timer (actual_Xxx_Y_Timer) is 
   // pre-loaded with the ON-DELAY time (TIME_XXX_Y_ON_DEL).
   // 
   // This prevents the alarm/warning from activating instantly, if the actual_Value is outside the
   // alarm/warning setpoint. This condition could arise because the timer is set to zero while ever
   // the alarm/warning is disabled.
   // 
   // Note:    Technically, the ENABLE bit should not be modified at run-time, it is stored in a static
   //      data block; however, the condition could arise if that static data block is being used
   //      as a recipe block. mask signals can of course be changed at run-time.
   // ▄▄▄▄▄▄▄▄▄▄▄▄▄▄▄▄▄▄▄▄▄▄▄▄▄▄▄▄▄▄▄▄▄▄▄▄▄▄▄▄▄▄▄▄
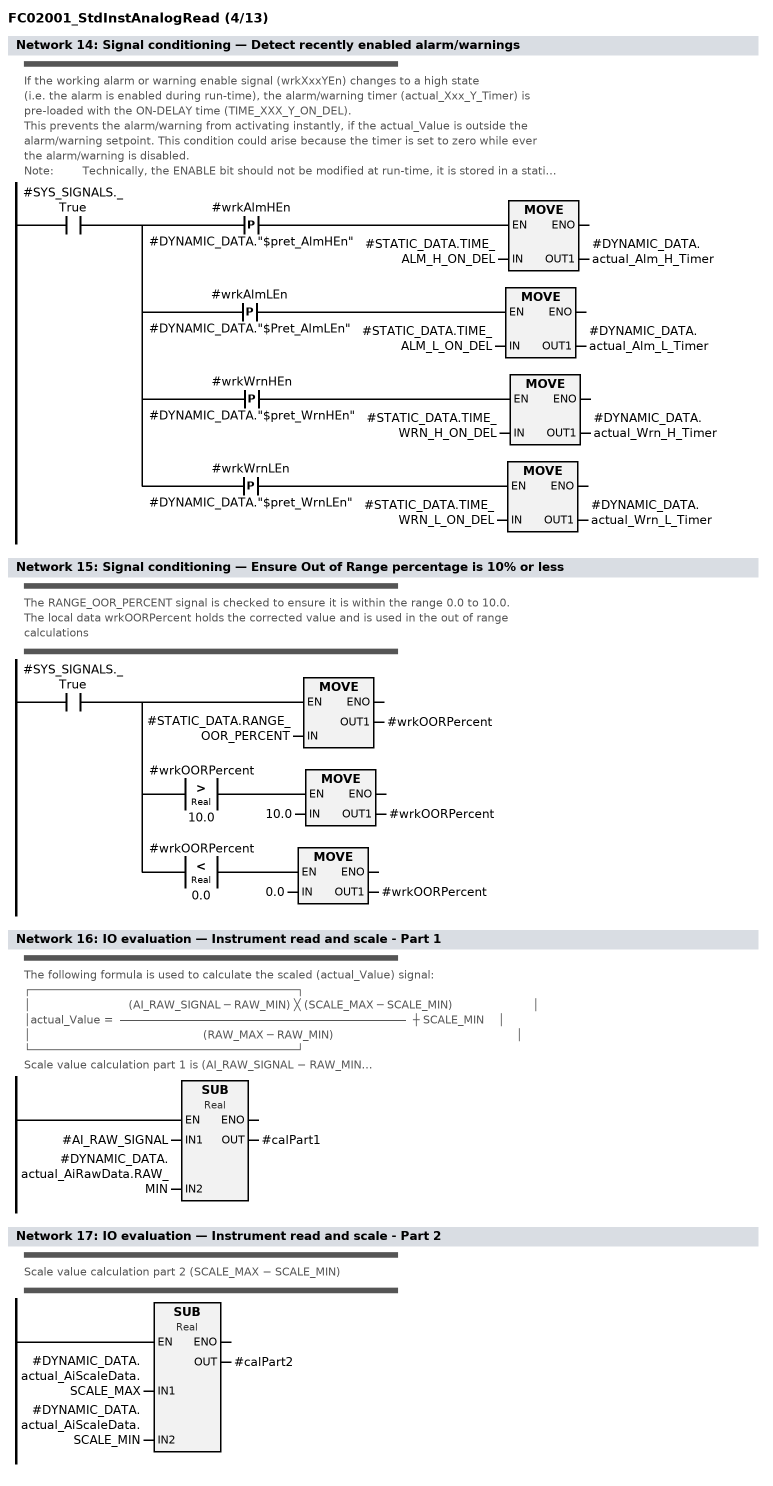
   RUNG wire#powerrail
      Contact( #SYS_SIGNALS._True )
      wire#w1
      P_Contact(operand := #wrkAlmHEn, bit := #DYNAMIC_DATA."$pret_AlmHEn")
      { S7_GenerateENO := "TRUE" } Move(in := #STATIC_DATA.TIME_ALM_H_ON_DEL, out1 => #DYNAMIC_DATA.actual_Alm_H_Timer)
   END_RUNG
   RUNG wire#w1
      P_Contact(operand := #wrkAlmLEn, bit := #DYNAMIC_DATA."$Pret_AlmLEn")
      { S7_GenerateENO := "TRUE" } Move(in := #STATIC_DATA.TIME_ALM_L_ON_DEL, out1 => #DYNAMIC_DATA.actual_Alm_L_Timer)
   END_RUNG
   RUNG wire#w1
      P_Contact(operand := #wrkWrnHEn, bit := #DYNAMIC_DATA."$pret_WrnHEn")
      { S7_GenerateENO := "TRUE" } Move(in := #STATIC_DATA.TIME_WRN_H_ON_DEL, out1 => #DYNAMIC_DATA.actual_Wrn_H_Timer)
   END_RUNG
   RUNG wire#w1
      P_Contact(operand := #wrkWrnLEn, bit := #DYNAMIC_DATA."$pret_WrnLEn")
      { S7_GenerateENO := "TRUE" } Move(in := #STATIC_DATA.TIME_WRN_L_ON_DEL, out1 => #DYNAMIC_DATA.actual_Wrn_L_Timer)
   END_RUNG
   // the same network as SCL:
   #_w1 := #SYS_SIGNALS._True AND #wrkAlmHEn AND NOT #DYNAMIC_DATA."$pret_AlmHEn";   // rising edge of #wrkAlmHEn
   #DYNAMIC_DATA."$pret_AlmHEn" := #wrkAlmHEn;
   IF #_w1 THEN #DYNAMIC_DATA.actual_Alm_H_Timer := #STATIC_DATA.TIME_ALM_H_ON_DEL; END_IF;
   #_w2 := #SYS_SIGNALS._True AND #wrkAlmLEn AND NOT #DYNAMIC_DATA."$Pret_AlmLEn";   // rising edge of #wrkAlmLEn
   #DYNAMIC_DATA."$Pret_AlmLEn" := #wrkAlmLEn;
   IF #_w2 THEN #DYNAMIC_DATA.actual_Alm_L_Timer := #STATIC_DATA.TIME_ALM_L_ON_DEL; END_IF;
   #_w3 := #SYS_SIGNALS._True AND #wrkWrnHEn AND NOT #DYNAMIC_DATA."$pret_WrnHEn";   // rising edge of #wrkWrnHEn
   #DYNAMIC_DATA."$pret_WrnHEn" := #wrkWrnHEn;
   IF #_w3 THEN #DYNAMIC_DATA.actual_Wrn_H_Timer := #STATIC_DATA.TIME_WRN_H_ON_DEL; END_IF;
   #_w4 := #SYS_SIGNALS._True AND #wrkWrnLEn AND NOT #DYNAMIC_DATA."$pret_WrnLEn";   // rising edge of #wrkWrnLEn
   #DYNAMIC_DATA."$pret_WrnLEn" := #wrkWrnLEn;
   IF #_w4 THEN #DYNAMIC_DATA.actual_Wrn_L_Timer := #STATIC_DATA.TIME_WRN_L_ON_DEL; END_IF;
END_REGION

REGION Network 15: Signal conditioning — Ensure Out of Range percentage is 10% or less
   // ▀▀▀▀▀▀▀▀▀▀▀▀▀▀▀▀▀▀▀▀▀▀▀▀▀▀▀▀▀▀▀▀▀▀▀▀▀▀▀▀▀▀▀▀
   // The RANGE_OOR_PERCENT signal is checked to ensure it is within the range 0.0 to 10.0.
   // 
   // The local data wrkOORPercent holds the corrected value and is used in the out of range 
   // calculations
   // ▄▄▄▄▄▄▄▄▄▄▄▄▄▄▄▄▄▄▄▄▄▄▄▄▄▄▄▄▄▄▄▄▄▄▄▄▄▄▄▄▄▄▄▄
   RUNG wire#powerrail
      Contact( #SYS_SIGNALS._True )
      wire#w1
      { S7_GenerateENO := "TRUE" } Move(in := #STATIC_DATA.RANGE_OOR_PERCENT, out1 => #wrkOORPercent)
   END_RUNG
   RUNG wire#w1
      { S7_Templates := "SrcType := Real" } GT_Contact(in1 := #wrkOORPercent, in2 := 10.0)
      { S7_GenerateENO := "TRUE" } Move(in := 10.0, out1 => #wrkOORPercent)
   END_RUNG
   RUNG wire#w1
      { S7_Templates := "SrcType := Real" } LT_Contact(in1 := #wrkOORPercent, in2 := 0.0)
      { S7_GenerateENO := "TRUE" } Move(in := 0.0, out1 => #wrkOORPercent)
   END_RUNG
   // the same network as SCL:
   IF #SYS_SIGNALS._True THEN #wrkOORPercent := #STATIC_DATA.RANGE_OOR_PERCENT; END_IF;
   IF #SYS_SIGNALS._True AND (#wrkOORPercent > 10.0) THEN #wrkOORPercent := 10.0; END_IF;
   IF #SYS_SIGNALS._True AND (#wrkOORPercent < 0.0) THEN #wrkOORPercent := 0.0; END_IF;
END_REGION

REGION Network 16: IO evaluation — Instrument read and scale - Part 1
   // ▀▀▀▀▀▀▀▀▀▀▀▀▀▀▀▀▀▀▀▀▀▀▀▀▀▀▀▀▀▀▀▀▀▀▀▀▀▀▀▀▀▀▀▀
   // The following formula is used to calculate the scaled (actual_Value) signal:
   // ┌─────────────────────────────────────────┐
   // │                            (AI_RAW_SIGNAL ─ RAW_MIN) ╳ (SCALE_MAX ─ SCALE_MIN)          │
   // │actual_Value =  ――――――――――――――――――――――――――  ┼ SCALE_MIN    │
   // │                              (RAW_MAX ─ RAW_MIN)                    │
   // └─────────────────────────────────────────┘
   // 
   // 
   // Scale value calculation part 1 is (AI_RAW_SIGNAL − RAW_MIN)
   // ▄▄▄▄▄▄▄▄▄▄▄▄▄▄▄▄▄▄▄▄▄▄▄▄▄▄▄▄▄▄▄▄▄▄▄▄▄▄▄▄▄▄▄▄
   RUNG wire#powerrail
      { S7_Templates := "SrcType := Real"; S7_GenerateENO := "TRUE" } Sub(in1 := #AI_RAW_SIGNAL, in2 := #DYNAMIC_DATA.actual_AiRawData.RAW_MIN, out => #calPart1)
   END_RUNG
   // the same network as SCL:
   #calPart1 := #AI_RAW_SIGNAL - #DYNAMIC_DATA.actual_AiRawData.RAW_MIN;
END_REGION

REGION Network 17: IO evaluation — Instrument read and scale - Part 2
   // ▀▀▀▀▀▀▀▀▀▀▀▀▀▀▀▀▀▀▀▀▀▀▀▀▀▀▀▀▀▀▀▀▀▀▀▀▀▀▀▀▀▀▀▀
   // Scale value calculation part 2 (SCALE_MAX − SCALE_MIN)
   // ▄▄▄▄▄▄▄▄▄▄▄▄▄▄▄▄▄▄▄▄▄▄▄▄▄▄▄▄▄▄▄▄▄▄▄▄▄▄▄▄▄▄▄▄
   RUNG wire#powerrail
      { S7_Templates := "SrcType := Real"; S7_GenerateENO := "TRUE" } Sub(in1 := #DYNAMIC_DATA.actual_AiScaleData.SCALE_MAX, in2 := #DYNAMIC_DATA.actual_AiScaleData.SCALE_MIN, out => #calPart2)
   END_RUNG
   // the same network as SCL:
   #calPart2 := #DYNAMIC_DATA.actual_AiScaleData.SCALE_MAX - #DYNAMIC_DATA.actual_AiScaleData.SCALE_MIN;
END_REGION

REGION Network 18: IO evaluation — Instrument read and scale - Part 3
   // ▀▀▀▀▀▀▀▀▀▀▀▀▀▀▀▀▀▀▀▀▀▀▀▀▀▀▀▀▀▀▀▀▀▀▀▀▀▀▀▀▀▀▀▀
   // Scale value calculation part 3 (RAW_MAX − RAW_MIN)
   // 
   // Note:    To prevent inconsistencies and divide by zero errors, if a configuration error is present
   //      (resulting from incorrect range data and indicated by status_ConfigError = TRUE), the
   //      denominator of the calculation (CalPart3) is set to 3.402823 × 1038 (i.e. a very large 
   //      number), the result of this is that the  actual_Value will equal RANGE_SCALE_MIN for 
   //      all permitted values of AI_RAW_SIGNAL.
   // ▄▄▄▄▄▄▄▄▄▄▄▄▄▄▄▄▄▄▄▄▄▄▄▄▄▄▄▄▄▄▄▄▄▄▄▄▄▄▄▄▄▄▄▄
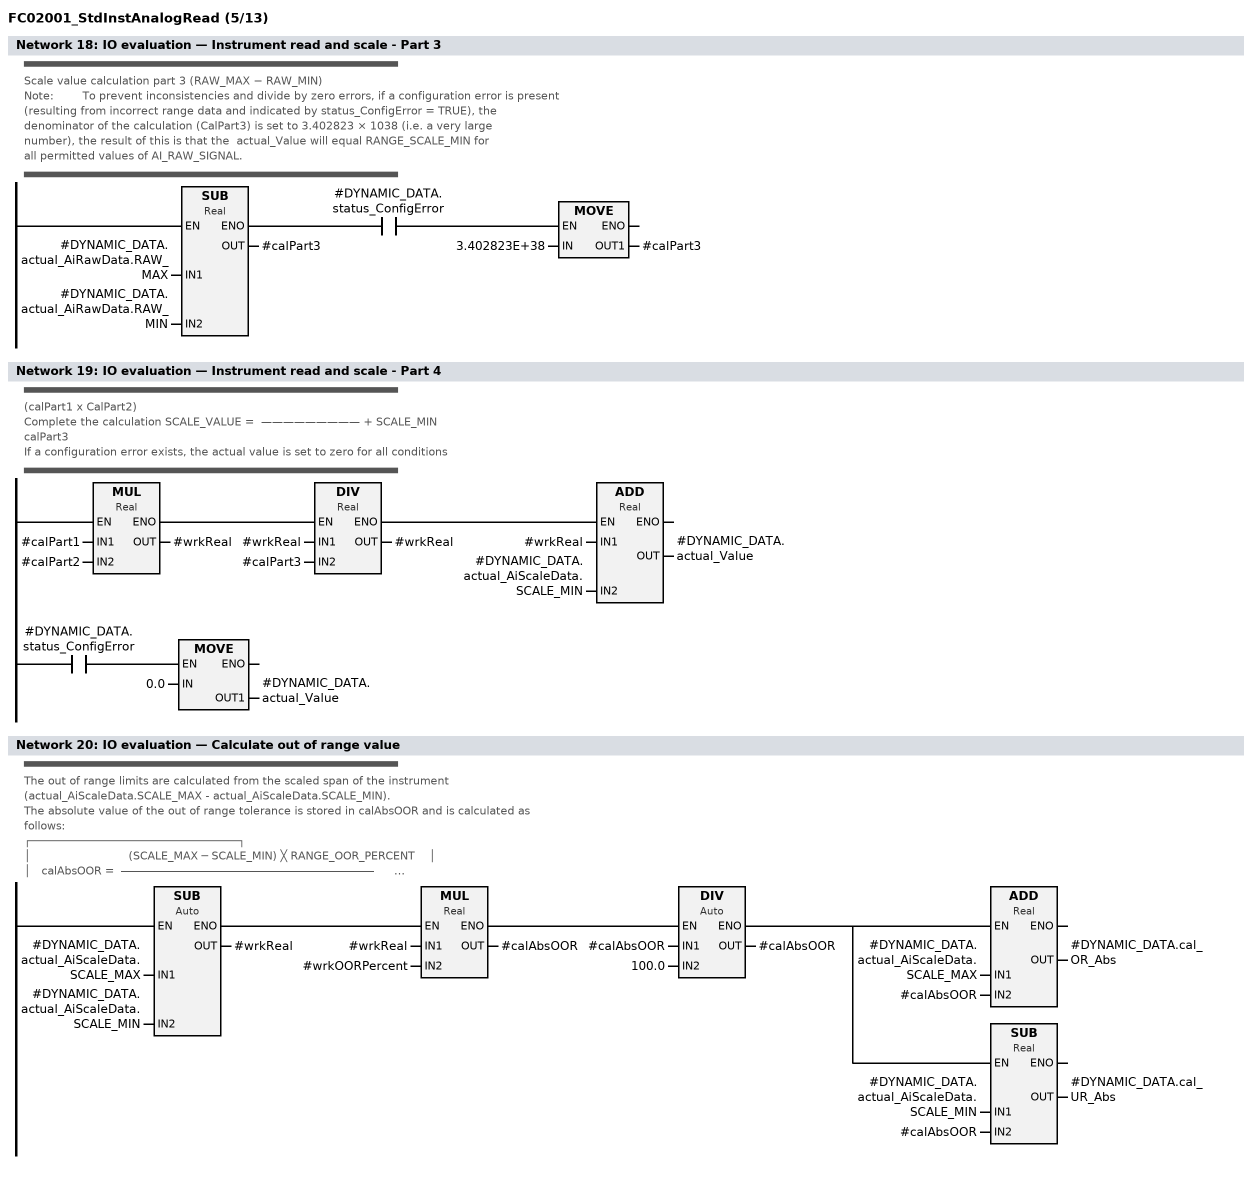
   RUNG wire#powerrail
      { S7_Templates := "SrcType := Real"; S7_GenerateENO := "TRUE" } Sub(in1 := #DYNAMIC_DATA.actual_AiRawData.RAW_MAX, in2 := #DYNAMIC_DATA.actual_AiRawData.RAW_MIN, out => #calPart3)
      Contact( #DYNAMIC_DATA.status_ConfigError )
      Move(in := 3.402823E+38, out1 => #calPart3)
   END_RUNG
   // the same network as SCL:
   // ENO of a box is taken as its EN; it also drops when the box reports an error
   #calPart3 := #DYNAMIC_DATA.actual_AiRawData.RAW_MAX - #DYNAMIC_DATA.actual_AiRawData.RAW_MIN;
   IF #DYNAMIC_DATA.status_ConfigError THEN #calPart3 := 3.402823E+38; END_IF;
END_REGION

REGION Network 19: IO evaluation — Instrument read and scale - Part 4
   // ▀▀▀▀▀▀▀▀▀▀▀▀▀▀▀▀▀▀▀▀▀▀▀▀▀▀▀▀▀▀▀▀▀▀▀▀▀▀▀▀▀▀▀▀
   //                                                                              (calPart1 x CalPart2)
   // Complete the calculation SCALE_VALUE =  ————————— + SCALE_MIN
   //                                                                                         calPart3
   // 
   // If a configuration error exists, the actual value is set to zero for all conditions
   // ▄▄▄▄▄▄▄▄▄▄▄▄▄▄▄▄▄▄▄▄▄▄▄▄▄▄▄▄▄▄▄▄▄▄▄▄▄▄▄▄▄▄▄▄
   RUNG wire#powerrail
      { S7_Templates := "SrcType := Real"; S7_GenerateENO := "TRUE" } Mul(in1 := #calPart1, in2 := #calPart2, out => #wrkReal)
      { S7_Templates := "SrcType := Real"; S7_GenerateENO := "TRUE" } Div(in1 := #wrkReal, in2 := #calPart3, out => #wrkReal)
      { S7_Templates := "SrcType := Real"; S7_GenerateENO := "TRUE" } Add(in1 := #wrkReal, in2 := #DYNAMIC_DATA.actual_AiScaleData.SCALE_MIN, out => #DYNAMIC_DATA.actual_Value)
   END_RUNG
   RUNG wire#powerrail
      Contact( #DYNAMIC_DATA.status_ConfigError )
      Move(in := 0.0, out1 => #DYNAMIC_DATA.actual_Value)
   END_RUNG
   // the same network as SCL:
   // ENO of a box is taken as its EN; it also drops when the box reports an error
   #wrkReal := #calPart1 * #calPart2;
   #wrkReal := #wrkReal / #calPart3;
   #DYNAMIC_DATA.actual_Value := #wrkReal + #DYNAMIC_DATA.actual_AiScaleData.SCALE_MIN;
   IF #DYNAMIC_DATA.status_ConfigError THEN #DYNAMIC_DATA.actual_Value := 0.0; END_IF;
END_REGION

REGION Network 20: IO evaluation — Calculate out of range value
   // ▀▀▀▀▀▀▀▀▀▀▀▀▀▀▀▀▀▀▀▀▀▀▀▀▀▀▀▀▀▀▀▀▀▀▀▀▀▀▀▀▀▀▀▀
   // The out of range limits are calculated from the scaled span of the instrument 
   // (actual_AiScaleData.SCALE_MAX - actual_AiScaleData.SCALE_MIN).
   // 
   // The absolute value of the out of range tolerance is stored in calAbsOOR and is calculated as
   // follows:
   // 
   // ┌────────────────────────────────┐
   // │                            (SCALE_MAX ─ SCALE_MIN) ╳ RANGE_OOR_PERCENT  │
   // │ calAbsOOR =  ―――――――――――――――――――――――    │
   // │                       100           │
   // └────────────────────────────────┘
   // 
   // The instrument is over range if the actual_Value is greater than SCALE_MAX + calcAbsOOR,
   // this absolute value is stored in the calculation variable cal_OR_Abs.
   // 
   // The instrument is under range if the AI_RAW_SIGNAL is less than SCALE_MIN - calcAbsOOR,
   // this absolute value is stored in the calculation variable cal_UR_Abs.
   // ▄▄▄▄▄▄▄▄▄▄▄▄▄▄▄▄▄▄▄▄▄▄▄▄▄▄▄▄▄▄▄▄▄▄▄▄▄▄▄▄▄▄▄▄
   RUNG wire#powerrail
      Sub(in1 := #DYNAMIC_DATA.actual_AiScaleData.SCALE_MAX, in2 := #DYNAMIC_DATA.actual_AiScaleData.SCALE_MIN, out => #wrkReal)
      { S7_Templates := "SrcType := Real"; S7_GenerateENO := "TRUE" } Mul(in1 := #wrkReal, in2 := #wrkOORPercent, out => #calAbsOOR)
      Div(in1 := #calAbsOOR, in2 := 100.0, out => #calAbsOOR)
      wire#w1
      { S7_Templates := "SrcType := Real"; S7_GenerateENO := "TRUE" } Add(in1 := #DYNAMIC_DATA.actual_AiScaleData.SCALE_MAX, in2 := #calAbsOOR, out => #DYNAMIC_DATA.cal_OR_Abs)
   END_RUNG
   RUNG wire#w1
      { S7_Templates := "SrcType := Real"; S7_GenerateENO := "TRUE" } Sub(in1 := #DYNAMIC_DATA.actual_AiScaleData.SCALE_MIN, in2 := #calAbsOOR, out => #DYNAMIC_DATA.cal_UR_Abs)
   END_RUNG
   // the same network as SCL:
   // ENO of a box is taken as its EN; it also drops when the box reports an error
   #wrkReal := #DYNAMIC_DATA.actual_AiScaleData.SCALE_MAX - #DYNAMIC_DATA.actual_AiScaleData.SCALE_MIN;
   #calAbsOOR := #wrkReal * #wrkOORPercent;
   #calAbsOOR := #calAbsOOR / 100.0;
   #DYNAMIC_DATA.cal_OR_Abs := #DYNAMIC_DATA.actual_AiScaleData.SCALE_MAX + #calAbsOOR;
   #DYNAMIC_DATA.cal_UR_Abs := #DYNAMIC_DATA.actual_AiScaleData.SCALE_MIN - #calAbsOOR;
END_REGION

REGION Network 21: IO evaluation — Out of range signals
   // ▀▀▀▀▀▀▀▀▀▀▀▀▀▀▀▀▀▀▀▀▀▀▀▀▀▀▀▀▀▀▀▀▀▀▀▀▀▀▀▀▀▀▀▀
   // The instrument is over range if the actual_Value is greater than or equal to cal_OR_Abs.
   // 
   // The instrument is under range if the actual_Value  is less than or equal to  cal_UR_Abs.
   // 
   // If either of these conditions is true, the common out of range signal is activated
   // 
   // Note:    The out of range signals are not generated if simulation mode is active
   // 
   // Note:    If the range information is incorrect (status_ConfigError = TRUE),
   //      Then all the out of range signals are activated msg_Flt_UnderRange, 
   //      msg_Flt_OverRange and msg_Flt_OutOfRange simultaneously, this is true even if
   //      simulation mode is active.
   // ▄▄▄▄▄▄▄▄▄▄▄▄▄▄▄▄▄▄▄▄▄▄▄▄▄▄▄▄▄▄▄▄▄▄▄▄▄▄▄▄▄▄▄▄
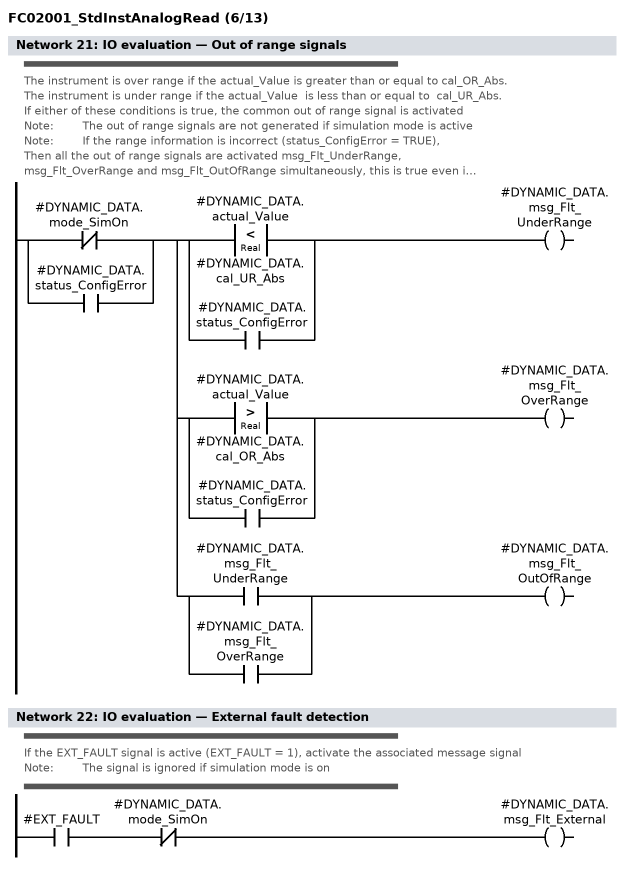
   RUNG wire#powerrail
      I_Contact( #DYNAMIC_DATA.mode_SimOn )
      wire#w1
      { S7_Templates := "SrcType := Real" } LT_Contact(in1 := #DYNAMIC_DATA.actual_Value, in2 := #DYNAMIC_DATA.cal_UR_Abs)
      wire#w2
      Coil( #DYNAMIC_DATA.msg_Flt_UnderRange )
   END_RUNG
   RUNG wire#powerrail
      Contact( #DYNAMIC_DATA.status_ConfigError )
   END_RUNG wire#w1
   RUNG wire#w1
      Contact( #DYNAMIC_DATA.status_ConfigError )
   END_RUNG wire#w2
   RUNG wire#w1
      { S7_Templates := "SrcType := Real" } GT_Contact(in1 := #DYNAMIC_DATA.actual_Value, in2 := #DYNAMIC_DATA.cal_OR_Abs)
      wire#w3
      Coil( #DYNAMIC_DATA.msg_Flt_OverRange )
   END_RUNG
   RUNG wire#w1
      Contact( #DYNAMIC_DATA.status_ConfigError )
   END_RUNG wire#w3
   RUNG wire#w1
      Contact( #DYNAMIC_DATA.msg_Flt_UnderRange )
      wire#w4
      Coil( #DYNAMIC_DATA.msg_Flt_OutOfRange )
   END_RUNG
   RUNG wire#w1
      Contact( #DYNAMIC_DATA.msg_Flt_OverRange )
   END_RUNG wire#w4
   // the same network as SCL:
   #_w1 := NOT #DYNAMIC_DATA.mode_SimOn OR #DYNAMIC_DATA.status_ConfigError;
   #DYNAMIC_DATA.msg_Flt_UnderRange := #_w1 AND ((#DYNAMIC_DATA.actual_Value < #DYNAMIC_DATA.cal_UR_Abs) OR #DYNAMIC_DATA.status_ConfigError);
   #DYNAMIC_DATA.msg_Flt_OverRange := #_w1 AND ((#DYNAMIC_DATA.actual_Value > #DYNAMIC_DATA.cal_OR_Abs) OR #DYNAMIC_DATA.status_ConfigError);
   #DYNAMIC_DATA.msg_Flt_OutOfRange := #_w1 AND (#DYNAMIC_DATA.msg_Flt_UnderRange OR #DYNAMIC_DATA.msg_Flt_OverRange);
END_REGION

REGION Network 22: IO evaluation — External fault detection
   // ▀▀▀▀▀▀▀▀▀▀▀▀▀▀▀▀▀▀▀▀▀▀▀▀▀▀▀▀▀▀▀▀▀▀▀▀▀▀▀▀▀▀▀▀
   // If the EXT_FAULT signal is active (EXT_FAULT = 1), activate the associated message signal
   // 
   // Note:    The signal is ignored if simulation mode is on
   // ▄▄▄▄▄▄▄▄▄▄▄▄▄▄▄▄▄▄▄▄▄▄▄▄▄▄▄▄▄▄▄▄▄▄▄▄▄▄▄▄▄▄▄▄
   RUNG wire#powerrail
      Contact( #EXT_FAULT )
      I_Contact( #DYNAMIC_DATA.mode_SimOn )
      Coil( #DYNAMIC_DATA.msg_Flt_External )
   END_RUNG
   // the same network as SCL:
   #DYNAMIC_DATA.msg_Flt_External := #EXT_FAULT AND NOT #DYNAMIC_DATA.mode_SimOn;
END_REGION

REGION Network 23: Operating mode — Simulation mode
   // ▀▀▀▀▀▀▀▀▀▀▀▀▀▀▀▀▀▀▀▀▀▀▀▀▀▀▀▀▀▀▀▀▀▀▀▀▀▀▀▀▀▀▀▀
   // If simulation mode is enabled (mode_SimOn = 1) and a configuration error is not present,
   // (status_ConfigError = 0) overwrite the actual_Value with the mode_SimValue signal set by the 
   // operator.
   // 
   // Note:    Any fault signals will be suppressed (turned off) is simulation mode is active
   //      and a configuration error is not present
   // 
   //      The simulated value (mode_SimValue) is restricted to the range given in 
   //      actual_AiScaleData.SCALE_MIN and actual_AiScaleData.SCALE_MAX
   // ▄▄▄▄▄▄▄▄▄▄▄▄▄▄▄▄▄▄▄▄▄▄▄▄▄▄▄▄▄▄▄▄▄▄▄▄▄▄▄▄▄▄▄▄
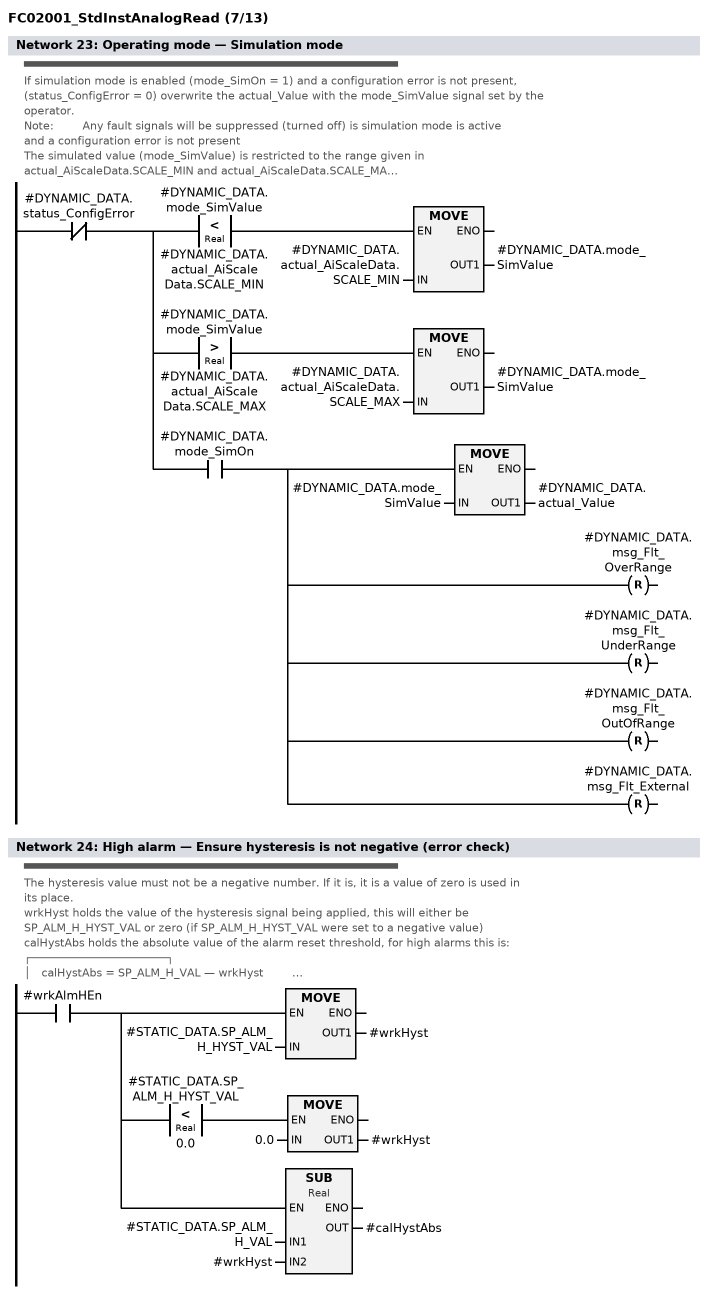
   RUNG wire#powerrail
      I_Contact( #DYNAMIC_DATA.status_ConfigError )
      wire#w1
      { S7_Templates := "SrcType := Real" } LT_Contact(in1 := #DYNAMIC_DATA.mode_SimValue, in2 := #DYNAMIC_DATA.actual_AiScaleData.SCALE_MIN)
      { S7_GenerateENO := "TRUE" } Move(in := #DYNAMIC_DATA.actual_AiScaleData.SCALE_MIN, out1 => #DYNAMIC_DATA.mode_SimValue)
   END_RUNG
   RUNG wire#w1
      { S7_Templates := "SrcType := Real" } GT_Contact(in1 := #DYNAMIC_DATA.mode_SimValue, in2 := #DYNAMIC_DATA.actual_AiScaleData.SCALE_MAX)
      { S7_GenerateENO := "TRUE" } Move(in := #DYNAMIC_DATA.actual_AiScaleData.SCALE_MAX, out1 => #DYNAMIC_DATA.mode_SimValue)
   END_RUNG
   RUNG wire#w1
      Contact( #DYNAMIC_DATA.mode_SimOn )
      wire#w2
      { S7_GenerateENO := "TRUE" } Move(in := #DYNAMIC_DATA.mode_SimValue, out1 => #DYNAMIC_DATA.actual_Value)
   END_RUNG
   RUNG wire#w2
      R_Coil( #DYNAMIC_DATA.msg_Flt_OverRange )
   END_RUNG
   RUNG wire#w2
      R_Coil( #DYNAMIC_DATA.msg_Flt_UnderRange )
   END_RUNG
   RUNG wire#w2
      R_Coil( #DYNAMIC_DATA.msg_Flt_OutOfRange )
   END_RUNG
   RUNG wire#w2
      R_Coil( #DYNAMIC_DATA.msg_Flt_External )
   END_RUNG
   // the same network as SCL:
   #_w1 := NOT #DYNAMIC_DATA.status_ConfigError;
   IF #_w1 AND (#DYNAMIC_DATA.mode_SimValue < #DYNAMIC_DATA.actual_AiScaleData.SCALE_MIN) THEN
       #DYNAMIC_DATA.mode_SimValue := #DYNAMIC_DATA.actual_AiScaleData.SCALE_MIN;
   END_IF;
   IF #_w1 AND (#DYNAMIC_DATA.mode_SimValue > #DYNAMIC_DATA.actual_AiScaleData.SCALE_MAX) THEN
       #DYNAMIC_DATA.mode_SimValue := #DYNAMIC_DATA.actual_AiScaleData.SCALE_MAX;
   END_IF;
   IF #_w1 AND #DYNAMIC_DATA.mode_SimOn THEN
       #DYNAMIC_DATA.actual_Value := #DYNAMIC_DATA.mode_SimValue;
       #DYNAMIC_DATA.msg_Flt_OverRange := FALSE;
       #DYNAMIC_DATA.msg_Flt_UnderRange := FALSE;
       #DYNAMIC_DATA.msg_Flt_OutOfRange := FALSE;
       #DYNAMIC_DATA.msg_Flt_External := FALSE;
   END_IF;
END_REGION

REGION Network 24: High alarm — Ensure hysteresis is not negative (error check)
   // ▀▀▀▀▀▀▀▀▀▀▀▀▀▀▀▀▀▀▀▀▀▀▀▀▀▀▀▀▀▀▀▀▀▀▀▀▀▀▀▀▀▀▀▀
   // The hysteresis value must not be a negative number. If it is, it is a value of zero is used in
   // its place.
   // 
   // wrkHyst holds the value of the hysteresis signal being applied, this will either be 
   // SP_ALM_H_HYST_VAL or zero (if SP_ALM_H_HYST_VAL were set to a negative value)
   // 
   // calHystAbs holds the absolute value of the alarm reset threshold, for high alarms this is:
   // ┌─────────────────────┐
   // │ calHystAbs = SP_ALM_H_VAL — wrkHyst      │
   // └─────────────────────┘
   // 
   // The two threshold values for the high alarm are thus:
   // 
   //      High alarm activation threshold = SP_ALM_H_VAL
   //      High alarm reset threshold          = calHystAbs
   // 
   // Note:    The hysteresis is only checked if alarm is being evaluated
   // ▄▄▄▄▄▄▄▄▄▄▄▄▄▄▄▄▄▄▄▄▄▄▄▄▄▄▄▄▄▄▄▄▄▄▄▄▄▄▄▄▄▄▄▄
   RUNG wire#powerrail
      Contact( #wrkAlmHEn )
      wire#w1
      { S7_GenerateENO := "TRUE" } Move(in := #STATIC_DATA.SP_ALM_H_HYST_VAL, out1 => #wrkHyst)
   END_RUNG
   RUNG wire#w1
      { S7_Templates := "SrcType := Real" } LT_Contact(in1 := #STATIC_DATA.SP_ALM_H_HYST_VAL, in2 := 0.0)
      { S7_GenerateENO := "TRUE" } Move(in := 0.0, out1 => #wrkHyst)
   END_RUNG
   RUNG wire#w1
      { S7_Templates := "SrcType := Real"; S7_GenerateENO := "TRUE" } Sub(in1 := #STATIC_DATA.SP_ALM_H_VAL, in2 := #wrkHyst, out => #calHystAbs)
   END_RUNG
   // the same network as SCL:
   IF #wrkAlmHEn THEN #wrkHyst := #STATIC_DATA.SP_ALM_H_HYST_VAL; END_IF;
   IF #wrkAlmHEn AND (#STATIC_DATA.SP_ALM_H_HYST_VAL < 0.0) THEN #wrkHyst := 0.0; END_IF;
   IF #wrkAlmHEn THEN #calHystAbs := #STATIC_DATA.SP_ALM_H_VAL - #wrkHyst; END_IF;
END_REGION

